  PROC DrawPart107()
    MoveL Offs(pOrigin,356.52,241.10,0.00),v60,z0,tPen\WObj:=wPaper;
    MoveL Offs(pOrigin,353.06,244.55,0.00),v40,z0,tPen\WObj:=wPaper;
    MoveL Offs(pOrigin,352.89,244.16,0.00),v40,z0,tPen\WObj:=wPaper;
    MoveL Offs(pOrigin,351.08,242.36,0.00),v40,z0,tPen\WObj:=wPaper;
    MoveL Offs(pOrigin,351.27,241.86,0.00),v40,z0,tPen\WObj:=wPaper;
    MoveL Offs(pOrigin,347.97,245.17,0.00),v40,z0,tPen\WObj:=wPaper;
    MoveL Offs(pOrigin,347.50,244.74,0.00),v40,z0,tPen\WObj:=wPaper;
    MoveL Offs(pOrigin,345.69,242.94,0.00),v40,z0,tPen\WObj:=wPaper;
    MoveL Offs(pOrigin,346.48,242.18,0.00),v40,z0,tPen\WObj:=wPaper;
    MoveL Offs(pOrigin,343.17,245.48,0.00),v40,z0,tPen\WObj:=wPaper;
    MoveL Offs(pOrigin,343.30,245.03,0.00),v40,z0,tPen\WObj:=wPaper;
    MoveL Offs(pOrigin,341.65,243.38,0.00),v40,z0,tPen\WObj:=wPaper;
    MoveL Offs(pOrigin,341.53,242.64,0.00),v40,z0,tPen\WObj:=wPaper;
    MoveL Offs(pOrigin,338.23,245.95,0.00),v40,z0,tPen\WObj:=wPaper;
    MoveL Offs(pOrigin,338.06,245.76,0.00),v40,z0,tPen\WObj:=wPaper;
    MoveL Offs(pOrigin,336.26,243.96,0.00),v40,z0,tPen\WObj:=wPaper;
    MoveL Offs(pOrigin,336.59,243.10,0.00),v40,z0,tPen\WObj:=wPaper;
    MoveL Offs(pOrigin,333.58,246.11,0.00),v40,z0,tPen\WObj:=wPaper;
    MoveL Offs(pOrigin,333.72,245.90,0.00),v40,z0,tPen\WObj:=wPaper;
    MoveL Offs(pOrigin,331.91,244.10,0.00),v40,z0,tPen\WObj:=wPaper;
    MoveL Offs(pOrigin,331.64,243.57,0.00),v40,z0,tPen\WObj:=wPaper;
    MoveL Offs(pOrigin,328.64,246.57,0.00),v40,z0,tPen\WObj:=wPaper;
    MoveL Offs(pOrigin,328.18,246.33,0.00),v40,z0,tPen\WObj:=wPaper;
    MoveL Offs(pOrigin,326.37,244.53,0.00),v40,fine,tPen\WObj:=wPaper;
    MoveL Offs(pOrigin,326.37,244.53,6.00),v60,z5,tPen\WObj:=wPaper;
    MoveL Offs(pOrigin,325.18,246.32,6.00),vTravel,z5,tPen\WObj:=wPaper;
    MoveL Offs(pOrigin,325.18,246.32,0.00),v60,z0,tPen\WObj:=wPaper;
    MoveL Offs(pOrigin,323.38,244.52,0.00),v40,z0,tPen\WObj:=wPaper;
    MoveL Offs(pOrigin,324.00,243.74,0.00),v40,z0,tPen\WObj:=wPaper;
    MoveL Offs(pOrigin,320.70,247.05,0.00),v40,z0,tPen\WObj:=wPaper;
    MoveL Offs(pOrigin,320.84,246.46,0.00),v40,z0,tPen\WObj:=wPaper;
    MoveL Offs(pOrigin,319.18,244.81,0.00),v40,z0,tPen\WObj:=wPaper;
    MoveL Offs(pOrigin,319.36,243.91,0.00),v40,z0,tPen\WObj:=wPaper;
    MoveL Offs(pOrigin,316.20,247.06,0.00),v40,z0,tPen\WObj:=wPaper;
    MoveL Offs(pOrigin,316.64,246.75,0.00),v40,z0,tPen\WObj:=wPaper;
    MoveL Offs(pOrigin,314.69,244.79,0.00),v40,z0,tPen\WObj:=wPaper;
    MoveL Offs(pOrigin,314.56,244.22,0.00),v40,z0,tPen\WObj:=wPaper;
    MoveL Offs(pOrigin,311.56,247.23,0.00),v40,z0,tPen\WObj:=wPaper;
    MoveL Offs(pOrigin,312.15,246.73,0.00),v40,z0,tPen\WObj:=wPaper;
    MoveL Offs(pOrigin,310.35,244.93,0.00),v40,z0,tPen\WObj:=wPaper;
    MoveL Offs(pOrigin,310.07,244.23,0.00),v40,z0,tPen\WObj:=wPaper;
    MoveL Offs(pOrigin,307.06,247.24,0.00),v40,z0,tPen\WObj:=wPaper;
    MoveL Offs(pOrigin,307.66,246.72,0.00),v40,z0,tPen\WObj:=wPaper;
    MoveL Offs(pOrigin,305.85,244.92,0.00),v40,z0,tPen\WObj:=wPaper;
    MoveL Offs(pOrigin,305.58,244.25,0.00),v40,z0,tPen\WObj:=wPaper;
    MoveL Offs(pOrigin,302.57,247.25,0.00),v40,z0,tPen\WObj:=wPaper;
    MoveL Offs(pOrigin,303.16,246.70,0.00),v40,z0,tPen\WObj:=wPaper;
    MoveL Offs(pOrigin,301.21,244.75,0.00),v40,z0,tPen\WObj:=wPaper;
    MoveL Offs(pOrigin,301.08,244.26,0.00),v40,z0,tPen\WObj:=wPaper;
    MoveL Offs(pOrigin,297.32,248.02,0.00),v40,z0,tPen\WObj:=wPaper;
    MoveL Offs(pOrigin,297.77,247.29,0.00),v40,z0,tPen\WObj:=wPaper;
    MoveL Offs(pOrigin,300.17,249.69,0.00),v40,z0,tPen\WObj:=wPaper;
    MoveL Offs(pOrigin,300.62,249.21,0.00),v40,z0,tPen\WObj:=wPaper;
    MoveL Offs(pOrigin,296.41,253.41,0.00),v40,z0,tPen\WObj:=wPaper;
    MoveL Offs(pOrigin,296.86,254.46,0.00),v40,z0,tPen\WObj:=wPaper;
    MoveL Offs(pOrigin,300.76,250.56,0.00),v40,z0,tPen\WObj:=wPaper;
    MoveL Offs(pOrigin,300.63,251.64,0.00),v40,z0,tPen\WObj:=wPaper;
    MoveL Offs(pOrigin,298.23,249.24,0.00),v40,fine,tPen\WObj:=wPaper;
    MoveL Offs(pOrigin,298.23,249.24,6.00),v60,z5,tPen\WObj:=wPaper;
    MoveL Offs(pOrigin,298.68,251.19,6.00),vTravel,z5,tPen\WObj:=wPaper;
    MoveL Offs(pOrigin,298.68,251.19,0.00),v60,z0,tPen\WObj:=wPaper;
    MoveL Offs(pOrigin,301.09,253.59,0.00),v40,z0,tPen\WObj:=wPaper;
    MoveL Offs(pOrigin,301.20,253.10,0.00),v40,z0,tPen\WObj:=wPaper;
    MoveL Offs(pOrigin,297.15,257.16,0.00),v40,z0,tPen\WObj:=wPaper;
    MoveL Offs(pOrigin,297.80,257.77,0.00),v40,z0,tPen\WObj:=wPaper;
    MoveL Offs(pOrigin,298.55,258.52,0.00),v40,z0,tPen\WObj:=wPaper;
    MoveL Offs(pOrigin,298.24,258.51,0.00),v40,z0,tPen\WObj:=wPaper;
    MoveL Offs(pOrigin,297.81,258.09,0.00),v40,z0,tPen\WObj:=wPaper;
    MoveL Offs(pOrigin,298.02,256.60,0.00),v40,fine,tPen\WObj:=wPaper;
    MoveL Offs(pOrigin,298.02,256.60,6.00),v60,z5,tPen\WObj:=wPaper;
    MoveL Offs(pOrigin,297.15,255.66,6.00),vTravel,z5,tPen\WObj:=wPaper;
    MoveL Offs(pOrigin,297.15,255.66,0.00),v60,z0,tPen\WObj:=wPaper;
    MoveL Offs(pOrigin,301.06,251.75,0.00),v40,fine,tPen\WObj:=wPaper;
    MoveL Offs(pOrigin,301.06,251.75,6.00),v60,z5,tPen\WObj:=wPaper;
    MoveL Offs(pOrigin,301.65,254.15,6.00),vTravel,z5,tPen\WObj:=wPaper;
    MoveL Offs(pOrigin,301.65,254.15,0.00),v60,z0,tPen\WObj:=wPaper;
    MoveL Offs(pOrigin,297.14,258.66,0.00),v40,fine,tPen\WObj:=wPaper;
    MoveL Offs(pOrigin,297.14,258.66,6.00),v60,z5,tPen\WObj:=wPaper;
    MoveL Offs(pOrigin,297.14,260.15,6.00),vTravel,z5,tPen\WObj:=wPaper;
    MoveL Offs(pOrigin,297.14,260.15,0.00),v60,z0,tPen\WObj:=wPaper;
    MoveL Offs(pOrigin,301.80,255.50,0.00),v40,z0,tPen\WObj:=wPaper;
    MoveL Offs(pOrigin,301.09,255.09,0.00),v40,z0,tPen\WObj:=wPaper;
    MoveL Offs(pOrigin,298.69,252.68,0.00),v40,fine,tPen\WObj:=wPaper;
    MoveL Offs(pOrigin,298.69,252.68,6.00),v60,z5,tPen\WObj:=wPaper;
    MoveL Offs(pOrigin,299.14,254.63,6.00),vTravel,z5,tPen\WObj:=wPaper;
    MoveL Offs(pOrigin,299.14,254.63,0.00),v60,z0,tPen\WObj:=wPaper;
    MoveL Offs(pOrigin,301.70,257.19,0.00),v40,z0,tPen\WObj:=wPaper;
    MoveL Offs(pOrigin,302.24,256.54,0.00),v40,z0,tPen\WObj:=wPaper;
    MoveL Offs(pOrigin,296.83,261.95,0.00),v40,fine,tPen\WObj:=wPaper;
    MoveL Offs(pOrigin,296.83,261.95,6.00),v60,z5,tPen\WObj:=wPaper;
    MoveL Offs(pOrigin,296.53,263.75,6.00),vTravel,z5,tPen\WObj:=wPaper;
    MoveL Offs(pOrigin,296.53,263.75,0.00),v60,z0,tPen\WObj:=wPaper;
    MoveL Offs(pOrigin,302.54,257.74,0.00),v40,fine,tPen\WObj:=wPaper;
    MoveL Offs(pOrigin,302.54,257.74,6.00),v60,z5,tPen\WObj:=wPaper;
    MoveL Offs(pOrigin,302.83,258.94,6.00),vTravel,z5,tPen\WObj:=wPaper;
    MoveL Offs(pOrigin,302.83,258.94,0.00),v60,z0,tPen\WObj:=wPaper;
    MoveL Offs(pOrigin,298.93,262.84,0.00),v40,fine,tPen\WObj:=wPaper;
    MoveL Offs(pOrigin,298.93,262.84,6.00),v60,z5,tPen\WObj:=wPaper;
    MoveL Offs(pOrigin,299.22,264.04,6.00),vTravel,z5,tPen\WObj:=wPaper;
    MoveL Offs(pOrigin,299.22,264.04,0.00),v60,z0,tPen\WObj:=wPaper;
    MoveL Offs(pOrigin,303.28,259.98,0.00),v40,z0,tPen\WObj:=wPaper;
    MoveL Offs(pOrigin,302.45,259.44,0.00),v40,z0,tPen\WObj:=wPaper;
    MoveL Offs(pOrigin,299.60,256.58,0.00),v40,fine,tPen\WObj:=wPaper;
    MoveL Offs(pOrigin,299.60,256.58,6.00),v60,z5,tPen\WObj:=wPaper;
    MoveL Offs(pOrigin,300.35,258.83,6.00),vTravel,z5,tPen\WObj:=wPaper;
    MoveL Offs(pOrigin,300.35,258.83,0.00),v60,z0,tPen\WObj:=wPaper;
    MoveL Offs(pOrigin,303.06,261.53,0.00),v40,z0,tPen\WObj:=wPaper;
    MoveL Offs(pOrigin,303.58,261.18,0.00),v40,z0,tPen\WObj:=wPaper;
    MoveL Offs(pOrigin,298.77,265.99,0.00),v40,fine,tPen\WObj:=wPaper;
    MoveL Offs(pOrigin,298.77,265.99,6.00),v60,z5,tPen\WObj:=wPaper;
    MoveL Offs(pOrigin,297.42,264.35,6.00),vTravel,z5,tPen\WObj:=wPaper;
    MoveL Offs(pOrigin,297.42,264.35,0.00),v60,z0,tPen\WObj:=wPaper;
    MoveL Offs(pOrigin,296.52,265.25,0.00),v40,fine,tPen\WObj:=wPaper;
    MoveL Offs(pOrigin,296.52,265.25,6.00),v60,z5,tPen\WObj:=wPaper;
    MoveL Offs(pOrigin,295.69,268.08,6.00),vTravel,z5,tPen\WObj:=wPaper;
    MoveL Offs(pOrigin,295.69,268.08,0.00),v60,z0,tPen\WObj:=wPaper;
    MoveL Offs(pOrigin,297.95,260.21,0.00),v40,z0,tPen\WObj:=wPaper;
    MoveL Offs(pOrigin,298.45,259.79,0.00),v40,fine,tPen\WObj:=wPaper;
    MoveL Offs(pOrigin,298.45,259.79,6.00),v60,z5,tPen\WObj:=wPaper;
    MoveL Offs(pOrigin,301.11,261.08,6.00),vTravel,z5,tPen\WObj:=wPaper;
  ENDPROC

  PROC DrawPart108()
    MoveL Offs(pOrigin,301.11,261.08,0.00),v60,z0,tPen\WObj:=wPaper;
    MoveL Offs(pOrigin,303.21,263.18,0.00),v40,z0,tPen\WObj:=wPaper;
    MoveL Offs(pOrigin,303.72,262.53,0.00),v40,z0,tPen\WObj:=wPaper;
    MoveL Offs(pOrigin,297.86,268.39,0.00),v40,fine,tPen\WObj:=wPaper;
    MoveL Offs(pOrigin,297.86,268.39,6.00),v60,z5,tPen\WObj:=wPaper;
    MoveL Offs(pOrigin,296.51,269.74,6.00),vTravel,z5,tPen\WObj:=wPaper;
    MoveL Offs(pOrigin,296.51,269.74,0.00),v60,z0,tPen\WObj:=wPaper;
    MoveL Offs(pOrigin,294.56,271.70,0.00),v40,z0,tPen\WObj:=wPaper;
    MoveL Offs(pOrigin,293.80,272.45,0.00),v40,z0,tPen\WObj:=wPaper;
    MoveL Offs(pOrigin,278.33,287.92,0.00),v40,fine,tPen\WObj:=wPaper;
    MoveL Offs(pOrigin,278.33,287.92,6.00),v60,z5,tPen\WObj:=wPaper;
    MoveL Offs(pOrigin,278.62,289.12,6.00),vTravel,z5,tPen\WObj:=wPaper;
    MoveL Offs(pOrigin,278.62,289.12,0.00),v60,z0,tPen\WObj:=wPaper;
    MoveL Offs(pOrigin,294.70,273.04,0.00),v40,fine,tPen\WObj:=wPaper;
    MoveL Offs(pOrigin,294.70,273.04,6.00),v60,z5,tPen\WObj:=wPaper;
    MoveL Offs(pOrigin,295.90,273.34,6.00),vTravel,z5,tPen\WObj:=wPaper;
    MoveL Offs(pOrigin,295.90,273.34,0.00),v60,z0,tPen\WObj:=wPaper;
    MoveL Offs(pOrigin,278.62,290.62,0.00),v40,z0,tPen\WObj:=wPaper;
    MoveL Offs(pOrigin,279.63,290.37,0.00),v40,z0,tPen\WObj:=wPaper;
    MoveL Offs(pOrigin,286.24,296.99,0.00),v40,z0,tPen\WObj:=wPaper;
    MoveL Offs(pOrigin,285.27,297.19,0.00),v40,z0,tPen\WObj:=wPaper;
    MoveL Offs(pOrigin,283.58,297.19,0.00),v40,z0,tPen\WObj:=wPaper;
    MoveL Offs(pOrigin,283.58,297.19,0.00),v40,z0,tPen\WObj:=wPaper;
    MoveL Offs(pOrigin,282.09,300.38,0.00),v40,z0,tPen\WObj:=wPaper;
    MoveL Offs(pOrigin,282.73,300.59,0.00),v40,z0,tPen\WObj:=wPaper;
    MoveL Offs(pOrigin,285.70,298.04,0.00),v40,z0,tPen\WObj:=wPaper;
    MoveL Offs(pOrigin,285.27,297.19,0.00),v40,z0,tPen\WObj:=wPaper;
    MoveL Offs(pOrigin,285.70,295.06,0.00),v40,z0,tPen\WObj:=wPaper;
    MoveL Offs(pOrigin,287.19,294.42,0.00),v40,z0,tPen\WObj:=wPaper;
    MoveL Offs(pOrigin,287.19,294.42,0.00),v40,z0,tPen\WObj:=wPaper;
    MoveL Offs(pOrigin,288.89,295.06,0.00),v40,z0,tPen\WObj:=wPaper;
    MoveL Offs(pOrigin,289.31,295.06,0.00),v40,z0,tPen\WObj:=wPaper;
    MoveL Offs(pOrigin,289.52,294.42,0.00),v40,z0,tPen\WObj:=wPaper;
    MoveL Offs(pOrigin,290.59,294.42,0.00),v40,fine,tPen\WObj:=wPaper;
    MoveL Offs(pOrigin,290.59,294.42,6.00),v60,z5,tPen\WObj:=wPaper;
    MoveL Offs(pOrigin,290.16,295.70,6.00),vTravel,z5,tPen\WObj:=wPaper;
    MoveL Offs(pOrigin,290.16,295.70,0.00),v60,z0,tPen\WObj:=wPaper;
    MoveL Offs(pOrigin,289.31,295.06,0.00),v40,fine,tPen\WObj:=wPaper;
    MoveL Offs(pOrigin,289.31,295.06,6.00),v60,z5,tPen\WObj:=wPaper;
    MoveL Offs(pOrigin,290.80,295.90,6.00),vTravel,z5,tPen\WObj:=wPaper;
    MoveL Offs(pOrigin,290.80,295.90,0.00),v60,z0,tPen\WObj:=wPaper;
    MoveL Offs(pOrigin,297.18,295.90,0.00),v40,z0,tPen\WObj:=wPaper;
    MoveL Offs(pOrigin,297.62,296.42,0.00),v40,z0,tPen\WObj:=wPaper;
    MoveL Offs(pOrigin,280.19,278.99,0.00),v40,z0,tPen\WObj:=wPaper;
    MoveL Offs(pOrigin,280.91,278.91,0.00),v40,z0,tPen\WObj:=wPaper;
    MoveL Offs(pOrigin,280.91,281.25,0.00),v40,z0,tPen\WObj:=wPaper;
    MoveL Offs(pOrigin,280.60,282.17,0.00),v40,z0,tPen\WObj:=wPaper;
    MoveL Offs(pOrigin,288.68,282.17,0.00),v40,fine,tPen\WObj:=wPaper;
    MoveL Offs(pOrigin,288.68,282.17,6.00),v60,z5,tPen\WObj:=wPaper;
    MoveL Offs(pOrigin,287.25,281.04,6.00),vTravel,z5,tPen\WObj:=wPaper;
    MoveL Offs(pOrigin,287.25,281.04,0.00),v60,z0,tPen\WObj:=wPaper;
    MoveL Offs(pOrigin,287.25,279.76,0.00),v40,z0,tPen\WObj:=wPaper;
    MoveL Offs(pOrigin,286.98,279.00,0.00),v40,z0,tPen\WObj:=wPaper;
    MoveL Offs(pOrigin,291.44,279.00,0.00),v40,fine,tPen\WObj:=wPaper;
    MoveL Offs(pOrigin,291.44,279.00,6.00),v60,z5,tPen\WObj:=wPaper;
    MoveL Offs(pOrigin,292.50,278.27,6.00),vTravel,z5,tPen\WObj:=wPaper;
    MoveL Offs(pOrigin,292.50,278.27,0.00),v60,z0,tPen\WObj:=wPaper;
    MoveL Offs(pOrigin,291.86,277.28,0.00),v40,z0,tPen\WObj:=wPaper;
    MoveL Offs(pOrigin,290.16,277.00,0.00),v40,z0,tPen\WObj:=wPaper;
    MoveL Offs(pOrigin,290.38,276.36,0.00),v40,z0,tPen\WObj:=wPaper;
    MoveL Offs(pOrigin,291.01,276.15,0.00),v40,z0,tPen\WObj:=wPaper;
    MoveL Offs(pOrigin,291.47,276.58,0.00),v40,z0,tPen\WObj:=wPaper;
    MoveL Offs(pOrigin,291.47,275.09,0.00),v40,z0,tPen\WObj:=wPaper;
    MoveL Offs(pOrigin,291.47,274.02,0.00),v40,z0,tPen\WObj:=wPaper;
    MoveL Offs(pOrigin,291.47,272.32,0.00),v40,z0,tPen\WObj:=wPaper;
    MoveL Offs(pOrigin,291.44,271.61,0.00),v40,z0,tPen\WObj:=wPaper;
    MoveL Offs(pOrigin,283.58,271.61,0.00),v40,z0,tPen\WObj:=wPaper;
    MoveL Offs(pOrigin,283.15,272.33,0.00),v40,z0,tPen\WObj:=wPaper;
    MoveL Offs(pOrigin,282.09,273.17,0.00),v40,z0,tPen\WObj:=wPaper;
    MoveL Offs(pOrigin,282.09,273.17,0.00),v40,z0,tPen\WObj:=wPaper;
    MoveL Offs(pOrigin,280.39,273.17,0.00),v40,z0,tPen\WObj:=wPaper;
    MoveL Offs(pOrigin,279.75,272.75,0.00),v40,z0,tPen\WObj:=wPaper;
    MoveL Offs(pOrigin,280.17,273.00,0.00),v40,z0,tPen\WObj:=wPaper;
    MoveL Offs(pOrigin,275.82,268.64,0.00),v40,z0,tPen\WObj:=wPaper;
    MoveL Offs(pOrigin,275.24,268.61,0.00),v40,z0,tPen\WObj:=wPaper;
    MoveL Offs(pOrigin,277.49,266.36,0.00),v40,fine,tPen\WObj:=wPaper;
    MoveL Offs(pOrigin,277.49,266.36,6.00),v60,z5,tPen\WObj:=wPaper;
    MoveL Offs(pOrigin,277.64,267.70,6.00),vTravel,z5,tPen\WObj:=wPaper;
    MoveL Offs(pOrigin,277.64,267.70,0.00),v60,z0,tPen\WObj:=wPaper;
    MoveL Offs(pOrigin,274.79,270.56,0.00),v40,z0,tPen\WObj:=wPaper;
    MoveL Offs(pOrigin,275.50,271.48,0.00),v40,z0,tPen\WObj:=wPaper;
    MoveL Offs(pOrigin,274.86,271.90,0.00),v40,z0,tPen\WObj:=wPaper;
    MoveL Offs(pOrigin,274.44,273.39,0.00),v40,z0,tPen\WObj:=wPaper;
    MoveL Offs(pOrigin,274.44,273.39,0.00),v40,z0,tPen\WObj:=wPaper;
    MoveL Offs(pOrigin,272.10,274.45,0.00),v40,z0,tPen\WObj:=wPaper;
    MoveL Offs(pOrigin,270.40,274.66,0.00),v40,z0,tPen\WObj:=wPaper;
    MoveL Offs(pOrigin,269.76,274.38,0.00),v40,z0,tPen\WObj:=wPaper;
    MoveL Offs(pOrigin,268.49,274.45,0.00),v40,z0,tPen\WObj:=wPaper;
    MoveL Offs(pOrigin,268.49,274.45,0.00),v40,z0,tPen\WObj:=wPaper;
    MoveL Offs(pOrigin,267.64,275.44,0.00),v40,z0,tPen\WObj:=wPaper;
    MoveL Offs(pOrigin,264.45,276.36,0.00),v40,z0,tPen\WObj:=wPaper;
    MoveL Offs(pOrigin,264.45,276.36,0.00),v40,z0,tPen\WObj:=wPaper;
    MoveL Offs(pOrigin,264.02,277.00,0.00),v40,z0,tPen\WObj:=wPaper;
    MoveL Offs(pOrigin,263.39,277.00,0.00),v40,z0,tPen\WObj:=wPaper;
    MoveL Offs(pOrigin,263.17,276.36,0.00),v40,z0,tPen\WObj:=wPaper;
    MoveL Offs(pOrigin,263.17,276.36,0.00),v40,z0,tPen\WObj:=wPaper;
    MoveL Offs(pOrigin,264.45,276.15,0.00),v40,z0,tPen\WObj:=wPaper;
    MoveL Offs(pOrigin,264.45,276.36,0.00),v40,z0,tPen\WObj:=wPaper;
    MoveL Offs(pOrigin,264.15,276.40,0.00),v40,z0,tPen\WObj:=wPaper;
    MoveL Offs(pOrigin,259.50,271.74,0.00),v40,fine,tPen\WObj:=wPaper;
    MoveL Offs(pOrigin,259.50,271.74,6.00),v60,z5,tPen\WObj:=wPaper;
    MoveL Offs(pOrigin,260.41,272.66,6.00),vTravel,z5,tPen\WObj:=wPaper;
    MoveL Offs(pOrigin,260.41,272.66,0.00),v60,z0,tPen\WObj:=wPaper;
    MoveL Offs(pOrigin,256.38,272.66,0.00),v40,z0,tPen\WObj:=wPaper;
    MoveL Offs(pOrigin,256.38,271.61,0.00),v40,z0,tPen\WObj:=wPaper;
    MoveL Offs(pOrigin,253.19,271.61,0.00),v40,z0,tPen\WObj:=wPaper;
    MoveL Offs(pOrigin,253.40,272.66,0.00),v40,z0,tPen\WObj:=wPaper;
    MoveL Offs(pOrigin,249.36,272.66,0.00),v40,z0,tPen\WObj:=wPaper;
    MoveL Offs(pOrigin,249.15,272.75,0.00),v40,z0,tPen\WObj:=wPaper;
    MoveL Offs(pOrigin,249.79,272.18,0.00),v40,z0,tPen\WObj:=wPaper;
    MoveL Offs(pOrigin,250.43,272.11,0.00),v40,z0,tPen\WObj:=wPaper;
    MoveL Offs(pOrigin,259.35,274.24,0.00),v40,z0,tPen\WObj:=wPaper;
    MoveL Offs(pOrigin,262.33,274.66,0.00),v40,z0,tPen\WObj:=wPaper;
    MoveL Offs(pOrigin,265.73,274.45,0.00),v40,z0,tPen\WObj:=wPaper;
    MoveL Offs(pOrigin,265.73,274.45,0.00),v40,z0,tPen\WObj:=wPaper;
    MoveL Offs(pOrigin,266.58,274.66,0.00),v40,z0,tPen\WObj:=wPaper;
    MoveL Offs(pOrigin,266.79,275.51,0.00),v40,z0,tPen\WObj:=wPaper;
    MoveL Offs(pOrigin,266.40,275.65,0.00),v40,z0,tPen\WObj:=wPaper;
    MoveL Offs(pOrigin,263.39,272.65,0.00),v40,z0,tPen\WObj:=wPaper;
    MoveL Offs(pOrigin,263.10,271.79,0.00),v40,z0,tPen\WObj:=wPaper;
  ENDPROC

  PROC DrawPart109()
    MoveL Offs(pOrigin,258.89,276.00,0.00),v40,z0,tPen\WObj:=wPaper;
    MoveL Offs(pOrigin,259.21,275.93,0.00),v40,z0,tPen\WObj:=wPaper;
    MoveL Offs(pOrigin,252.60,269.32,0.00),v40,z0,tPen\WObj:=wPaper;
    MoveL Offs(pOrigin,252.12,268.29,0.00),v40,z0,tPen\WObj:=wPaper;
    MoveL Offs(pOrigin,252.55,268.71,0.00),v40,z0,tPen\WObj:=wPaper;
    MoveL Offs(pOrigin,252.12,268.29,0.00),v40,z0,tPen\WObj:=wPaper;
    MoveL Offs(pOrigin,251.42,268.53,0.00),v40,z0,tPen\WObj:=wPaper;
    MoveL Offs(pOrigin,256.83,263.12,0.00),v40,fine,tPen\WObj:=wPaper;
    MoveL Offs(pOrigin,256.83,263.12,6.00),v60,z5,tPen\WObj:=wPaper;
    MoveL Offs(pOrigin,258.33,263.12,6.00),vTravel,z5,tPen\WObj:=wPaper;
    MoveL Offs(pOrigin,258.33,263.12,0.00),v60,z0,tPen\WObj:=wPaper;
    MoveL Offs(pOrigin,247.06,274.39,0.00),v40,z0,tPen\WObj:=wPaper;
    MoveL Offs(pOrigin,246.31,273.64,0.00),v40,z0,tPen\WObj:=wPaper;
    MoveL Offs(pOrigin,250.22,269.73,0.00),v40,z0,tPen\WObj:=wPaper;
    MoveL Offs(pOrigin,249.17,269.29,0.00),v40,z0,tPen\WObj:=wPaper;
    MoveL Offs(pOrigin,245.87,272.59,0.00),v40,z0,tPen\WObj:=wPaper;
    MoveL Offs(pOrigin,246.81,272.96,0.00),v40,z0,tPen\WObj:=wPaper;
    MoveL Offs(pOrigin,247.24,273.60,0.00),v40,z0,tPen\WObj:=wPaper;
    MoveL Offs(pOrigin,248.73,274.24,0.00),v40,z0,tPen\WObj:=wPaper;
    MoveL Offs(pOrigin,249.15,274.24,0.00),v40,z0,tPen\WObj:=wPaper;
    MoveL Offs(pOrigin,250.21,275.09,0.00),v40,z0,tPen\WObj:=wPaper;
    MoveL Offs(pOrigin,250.85,275.09,0.00),v40,z0,tPen\WObj:=wPaper;
    MoveL Offs(pOrigin,251.06,274.45,0.00),v40,z0,tPen\WObj:=wPaper;
    MoveL Offs(pOrigin,251.06,274.45,0.00),v40,z0,tPen\WObj:=wPaper;
    MoveL Offs(pOrigin,250.21,273.81,0.00),v40,z0,tPen\WObj:=wPaper;
    MoveL Offs(pOrigin,249.15,273.60,0.00),v40,z0,tPen\WObj:=wPaper;
    MoveL Offs(pOrigin,249.15,272.75,0.00),v40,z0,tPen\WObj:=wPaper;
    MoveL Offs(pOrigin,248.73,272.11,0.00),v40,z0,tPen\WObj:=wPaper;
    MoveL Offs(pOrigin,248.94,271.05,0.00),v40,z0,tPen\WObj:=wPaper;
    MoveL Offs(pOrigin,250.64,270.62,0.00),v40,z0,tPen\WObj:=wPaper;
    MoveL Offs(pOrigin,251.27,270.84,0.00),v40,z0,tPen\WObj:=wPaper;
    MoveL Offs(pOrigin,251.27,270.84,0.00),v40,z0,tPen\WObj:=wPaper;
    MoveL Offs(pOrigin,251.91,271.62,0.00),v40,z0,tPen\WObj:=wPaper;
    MoveL Offs(pOrigin,254.25,272.33,0.00),v40,z0,tPen\WObj:=wPaper;
    MoveL Offs(pOrigin,262.33,273.81,0.00),v40,z0,tPen\WObj:=wPaper;
    MoveL Offs(pOrigin,265.09,273.81,0.00),v40,z0,tPen\WObj:=wPaper;
    MoveL Offs(pOrigin,265.73,274.45,0.00),v40,z0,tPen\WObj:=wPaper;
    MoveL Offs(pOrigin,265.09,274.78,0.00),v40,z0,tPen\WObj:=wPaper;
    MoveL Offs(pOrigin,255.74,274.78,0.00),v40,z0,tPen\WObj:=wPaper;
    MoveL Offs(pOrigin,255.76,275.47,0.00),v40,z0,tPen\WObj:=wPaper;
    MoveL Offs(pOrigin,250.95,270.66,0.00),v40,z0,tPen\WObj:=wPaper;
    MoveL Offs(pOrigin,251.27,270.84,0.00),v40,z0,tPen\WObj:=wPaper;
    MoveL Offs(pOrigin,254.04,270.62,0.00),v40,z0,tPen\WObj:=wPaper;
    MoveL Offs(pOrigin,254.04,270.20,0.00),v40,z0,tPen\WObj:=wPaper;
    MoveL Offs(pOrigin,250.78,267.01,0.00),v40,z0,tPen\WObj:=wPaper;
    MoveL Offs(pOrigin,250.43,266.16,0.00),v40,z0,tPen\WObj:=wPaper;
    MoveL Offs(pOrigin,250.64,265.74,0.00),v40,z0,tPen\WObj:=wPaper;
    MoveL Offs(pOrigin,250.64,265.74,0.00),v40,z0,tPen\WObj:=wPaper;
    MoveL Offs(pOrigin,251.91,266.02,0.00),v40,z0,tPen\WObj:=wPaper;
    MoveL Offs(pOrigin,252.55,267.44,0.00),v40,z0,tPen\WObj:=wPaper;
    MoveL Offs(pOrigin,253.19,267.93,0.00),v40,z0,tPen\WObj:=wPaper;
    MoveL Offs(pOrigin,254.25,268.08,0.00),v40,z0,tPen\WObj:=wPaper;
    MoveL Offs(pOrigin,254.04,267.65,0.00),v40,z0,tPen\WObj:=wPaper;
    MoveL Offs(pOrigin,254.25,268.08,0.00),v40,z0,tPen\WObj:=wPaper;
    MoveL Offs(pOrigin,254.04,267.65,0.00),v40,fine,tPen\WObj:=wPaper;
    MoveL Offs(pOrigin,254.04,267.65,6.00),v60,z5,tPen\WObj:=wPaper;
    MoveL Offs(pOrigin,253.82,269.56,6.00),vTravel,z5,tPen\WObj:=wPaper;
    MoveL Offs(pOrigin,253.82,269.56,0.00),v60,z0,tPen\WObj:=wPaper;
    MoveL Offs(pOrigin,254.46,268.29,0.00),v40,z0,tPen\WObj:=wPaper;
    MoveL Offs(pOrigin,253.82,266.80,0.00),v40,z0,tPen\WObj:=wPaper;
    MoveL Offs(pOrigin,253.19,266.23,0.00),v40,z0,tPen\WObj:=wPaper;
    MoveL Offs(pOrigin,252.12,265.95,0.00),v40,z0,tPen\WObj:=wPaper;
    MoveL Offs(pOrigin,252.12,265.27,0.00),v40,z0,tPen\WObj:=wPaper;
    MoveL Offs(pOrigin,253.82,265.27,0.00),v40,z0,tPen\WObj:=wPaper;
    MoveL Offs(pOrigin,254.46,265.74,0.00),v40,z0,tPen\WObj:=wPaper;
    MoveL Offs(pOrigin,254.89,266.16,0.00),v40,z0,tPen\WObj:=wPaper;
    MoveL Offs(pOrigin,254.46,265.74,0.00),v40,z0,tPen\WObj:=wPaper;
    MoveL Offs(pOrigin,254.83,265.58,0.00),v40,z0,tPen\WObj:=wPaper;
    MoveL Offs(pOrigin,253.18,263.93,0.00),v40,z0,tPen\WObj:=wPaper;
    MoveL Offs(pOrigin,252.34,264.25,0.00),v40,z0,tPen\WObj:=wPaper;
    MoveL Offs(pOrigin,251.91,263.68,0.00),v40,z0,tPen\WObj:=wPaper;
    MoveL Offs(pOrigin,250.64,263.68,0.00),v40,z0,tPen\WObj:=wPaper;
    MoveL Offs(pOrigin,250.43,264.25,0.00),v40,z0,tPen\WObj:=wPaper;
    MoveL Offs(pOrigin,250.64,265.74,0.00),v40,z0,tPen\WObj:=wPaper;
    MoveL Offs(pOrigin,250.43,265.74,0.00),v40,z0,tPen\WObj:=wPaper;
    MoveL Offs(pOrigin,249.79,265.10,0.00),v40,z0,tPen\WObj:=wPaper;
    MoveL Offs(pOrigin,249.15,264.89,0.00),v40,z0,tPen\WObj:=wPaper;
    MoveL Offs(pOrigin,250.21,265.74,0.00),v40,z0,tPen\WObj:=wPaper;
    MoveL Offs(pOrigin,250.21,265.74,0.00),v40,z0,tPen\WObj:=wPaper;
    MoveL Offs(pOrigin,249.15,266.66,0.00),v40,z0,tPen\WObj:=wPaper;
    MoveL Offs(pOrigin,248.58,266.73,0.00),v40,z0,tPen\WObj:=wPaper;
    MoveL Offs(pOrigin,248.30,265.52,0.00),v40,z0,tPen\WObj:=wPaper;
    MoveL Offs(pOrigin,249.15,264.89,0.00),v40,z0,tPen\WObj:=wPaper;
    MoveL Offs(pOrigin,249.15,264.89,0.00),v40,z0,tPen\WObj:=wPaper;
    MoveL Offs(pOrigin,247.88,262.76,0.00),v40,z0,tPen\WObj:=wPaper;
    MoveL Offs(pOrigin,248.73,261.06,0.00),v40,z0,tPen\WObj:=wPaper;
    MoveL Offs(pOrigin,250.00,259.79,0.00),v40,z0,tPen\WObj:=wPaper;
    MoveL Offs(pOrigin,250.00,258.73,0.00),v40,z0,tPen\WObj:=wPaper;
    MoveL Offs(pOrigin,249.15,257.88,0.00),v40,z0,tPen\WObj:=wPaper;
    MoveL Offs(pOrigin,249.15,258.30,0.00),v40,z0,tPen\WObj:=wPaper;
    MoveL Offs(pOrigin,248.30,259.79,0.00),v40,z0,tPen\WObj:=wPaper;
    MoveL Offs(pOrigin,248.51,261.06,0.00),v40,fine,tPen\WObj:=wPaper;
    MoveL Offs(pOrigin,248.51,261.06,6.00),v60,z5,tPen\WObj:=wPaper;
    MoveL Offs(pOrigin,249.58,261.82,6.00),vTravel,z5,tPen\WObj:=wPaper;
    MoveL Offs(pOrigin,249.58,261.82,0.00),v60,z0,tPen\WObj:=wPaper;
    MoveL Offs(pOrigin,246.87,259.12,0.00),v40,z0,tPen\WObj:=wPaper;
    MoveL Offs(pOrigin,246.06,258.96,0.00),v40,z0,tPen\WObj:=wPaper;
    MoveL Offs(pOrigin,250.87,254.15,0.00),v40,fine,tPen\WObj:=wPaper;
    MoveL Offs(pOrigin,250.87,254.15,6.00),v60,z5,tPen\WObj:=wPaper;
    MoveL Offs(pOrigin,253.42,253.10,6.00),vTravel,z5,tPen\WObj:=wPaper;
    MoveL Offs(pOrigin,253.42,253.10,0.00),v60,z0,tPen\WObj:=wPaper;
    MoveL Offs(pOrigin,245.00,261.51,0.00),v40,z0,tPen\WObj:=wPaper;
    MoveL Offs(pOrigin,245.39,262.11,0.00),v40,z0,tPen\WObj:=wPaper;
    MoveL Offs(pOrigin,250.65,267.37,0.00),v40,z0,tPen\WObj:=wPaper;
    MoveL Offs(pOrigin,250.68,267.79,0.00),v40,z0,tPen\WObj:=wPaper;
    MoveL Offs(pOrigin,257.74,260.72,0.00),v40,fine,tPen\WObj:=wPaper;
    MoveL Offs(pOrigin,257.74,260.72,6.00),v60,z5,tPen\WObj:=wPaper;
    MoveL Offs(pOrigin,259.09,259.37,6.00),vTravel,z5,tPen\WObj:=wPaper;
    MoveL Offs(pOrigin,259.09,259.37,0.00),v60,z0,tPen\WObj:=wPaper;
    MoveL Offs(pOrigin,259.99,258.47,0.00),v40,z0,tPen\WObj:=wPaper;
    MoveL Offs(pOrigin,258.95,258.02,0.00),v40,z0,tPen\WObj:=wPaper;
    MoveL Offs(pOrigin,249.63,267.34,0.00),v40,fine,tPen\WObj:=wPaper;
    MoveL Offs(pOrigin,249.63,267.34,6.00),v60,z5,tPen\WObj:=wPaper;
    MoveL Offs(pOrigin,248.43,267.04,6.00),vTravel,z5,tPen\WObj:=wPaper;
    MoveL Offs(pOrigin,248.43,267.04,0.00),v60,z0,tPen\WObj:=wPaper;
    MoveL Offs(pOrigin,257.30,258.18,0.00),v40,fine,tPen\WObj:=wPaper;
    MoveL Offs(pOrigin,257.30,258.18,6.00),v60,z5,tPen\WObj:=wPaper;
    MoveL Offs(pOrigin,255.20,258.78,6.00),vTravel,z5,tPen\WObj:=wPaper;
    MoveL Offs(pOrigin,255.20,258.78,0.00),v60,z0,tPen\WObj:=wPaper;
    MoveL Offs(pOrigin,243.33,270.65,0.00),v40,fine,tPen\WObj:=wPaper;
  ENDPROC

  PROC DrawPart110()
    MoveL Offs(pOrigin,243.33,270.65,6.00),v60,z5,tPen\WObj:=wPaper;
    MoveL Offs(pOrigin,243.63,268.86,6.00),vTravel,z5,tPen\WObj:=wPaper;
    MoveL Offs(pOrigin,243.63,268.86,0.00),v60,z0,tPen\WObj:=wPaper;
    MoveL Offs(pOrigin,252.65,259.84,0.00),v40,fine,tPen\WObj:=wPaper;
    MoveL Offs(pOrigin,252.65,259.84,6.00),v60,z5,tPen\WObj:=wPaper;
    MoveL Offs(pOrigin,252.12,261.70,6.00),vTravel,z5,tPen\WObj:=wPaper;
    MoveL Offs(pOrigin,252.12,261.70,0.00),v60,z0,tPen\WObj:=wPaper;
    MoveL Offs(pOrigin,252.34,261.20,0.00),v40,z0,tPen\WObj:=wPaper;
    MoveL Offs(pOrigin,254.68,259.93,0.00),v40,z0,tPen\WObj:=wPaper;
    MoveL Offs(pOrigin,259.35,258.51,0.00),v40,z0,tPen\WObj:=wPaper;
    MoveL Offs(pOrigin,262.54,258.51,0.00),v40,fine,tPen\WObj:=wPaper;
    MoveL Offs(pOrigin,262.54,258.51,6.00),v60,z5,tPen\WObj:=wPaper;
    MoveL Offs(pOrigin,261.26,260.85,6.00),vTravel,z5,tPen\WObj:=wPaper;
    MoveL Offs(pOrigin,261.26,260.85,0.00),v60,z0,tPen\WObj:=wPaper;
    MoveL Offs(pOrigin,256.16,261.49,0.00),v40,z0,tPen\WObj:=wPaper;
    MoveL Offs(pOrigin,252.98,262.55,0.00),v40,z0,tPen\WObj:=wPaper;
    MoveL Offs(pOrigin,252.41,262.48,0.00),v40,z0,tPen\WObj:=wPaper;
    MoveL Offs(pOrigin,251.91,261.77,0.00),v40,z0,tPen\WObj:=wPaper;
    MoveL Offs(pOrigin,250.85,261.91,0.00),v40,fine,tPen\WObj:=wPaper;
    MoveL Offs(pOrigin,250.85,261.91,6.00),v60,z5,tPen\WObj:=wPaper;
    MoveL Offs(pOrigin,250.55,260.45,6.00),vTravel,z5,tPen\WObj:=wPaper;
    MoveL Offs(pOrigin,250.55,260.45,0.00),v60,z0,tPen\WObj:=wPaper;
    MoveL Offs(pOrigin,242.28,268.71,0.00),v40,z0,tPen\WObj:=wPaper;
    MoveL Offs(pOrigin,242.26,267.94,0.00),v40,z0,tPen\WObj:=wPaper;
    MoveL Offs(pOrigin,240.30,265.99,0.00),v40,z0,tPen\WObj:=wPaper;
    MoveL Offs(pOrigin,240.05,264.97,0.00),v40,z0,tPen\WObj:=wPaper;
    MoveL Offs(pOrigin,233.59,271.43,0.00),v40,z0,tPen\WObj:=wPaper;
    MoveL Offs(pOrigin,233.21,271.48,0.00),v40,z0,tPen\WObj:=wPaper;
    MoveL Offs(pOrigin,231.94,271.90,0.00),v40,z0,tPen\WObj:=wPaper;
    MoveL Offs(pOrigin,231.30,271.26,0.00),v40,z0,tPen\WObj:=wPaper;
    MoveL Offs(pOrigin,232.08,271.20,0.00),v40,z0,tPen\WObj:=wPaper;
    MoveL Offs(pOrigin,222.77,261.89,0.00),v40,z0,tPen\WObj:=wPaper;
    MoveL Offs(pOrigin,223.22,262.10,0.00),v40,z0,tPen\WObj:=wPaper;
    MoveL Offs(pOrigin,228.96,262.10,0.00),v40,z0,tPen\WObj:=wPaper;
    MoveL Offs(pOrigin,228.96,261.91,0.00),v40,z0,tPen\WObj:=wPaper;
    MoveL Offs(pOrigin,227.90,262.12,0.00),v40,z0,tPen\WObj:=wPaper;
    MoveL Offs(pOrigin,228.11,261.91,0.00),v40,z0,tPen\WObj:=wPaper;
    MoveL Offs(pOrigin,228.11,264.46,0.00),v40,z0,tPen\WObj:=wPaper;
    MoveL Offs(pOrigin,228.32,265.10,0.00),v40,z0,tPen\WObj:=wPaper;
    MoveL Offs(pOrigin,226.84,265.10,0.00),v40,z0,tPen\WObj:=wPaper;
    MoveL Offs(pOrigin,226.41,265.74,0.00),v40,z0,tPen\WObj:=wPaper;
    MoveL Offs(pOrigin,225.99,265.27,0.00),v40,z0,tPen\WObj:=wPaper;
    MoveL Offs(pOrigin,232.36,265.27,0.00),v40,z0,tPen\WObj:=wPaper;
    MoveL Offs(pOrigin,232.81,265.96,0.00),v40,z0,tPen\WObj:=wPaper;
    MoveL Offs(pOrigin,226.80,259.95,0.00),v40,z0,tPen\WObj:=wPaper;
    MoveL Offs(pOrigin,226.44,259.17,0.00),v40,z0,tPen\WObj:=wPaper;
    MoveL Offs(pOrigin,215.47,270.14,0.00),v40,z0,tPen\WObj:=wPaper;
    MoveL Offs(pOrigin,216.05,270.11,0.00),v40,z0,tPen\WObj:=wPaper;
    MoveL Offs(pOrigin,213.50,267.55,0.00),v40,z0,tPen\WObj:=wPaper;
    MoveL Offs(pOrigin,213.88,267.86,0.00),v40,z0,tPen\WObj:=wPaper;
    MoveL Offs(pOrigin,214.30,268.57,0.00),v40,z0,tPen\WObj:=wPaper;
    MoveL Offs(pOrigin,217.06,270.41,0.00),v40,z0,tPen\WObj:=wPaper;
    MoveL Offs(pOrigin,216.36,270.74,0.00),v40,z0,tPen\WObj:=wPaper;
    MoveL Offs(pOrigin,227.63,259.47,0.00),v40,fine,tPen\WObj:=wPaper;
    MoveL Offs(pOrigin,227.63,259.47,6.00),v60,z5,tPen\WObj:=wPaper;
    MoveL Offs(pOrigin,226.41,259.15,6.00),vTravel,z5,tPen\WObj:=wPaper;
    MoveL Offs(pOrigin,226.41,259.15,0.00),v60,z0,tPen\WObj:=wPaper;
    MoveL Offs(pOrigin,223.65,258.94,0.00),v40,z0,tPen\WObj:=wPaper;
    MoveL Offs(pOrigin,223.23,259.15,0.00),v40,z0,tPen\WObj:=wPaper;
    MoveL Offs(pOrigin,222.87,260.00,0.00),v40,z0,tPen\WObj:=wPaper;
    MoveL Offs(pOrigin,224.07,260.85,0.00),v40,z0,tPen\WObj:=wPaper;
    MoveL Offs(pOrigin,224.07,260.85,0.00),v40,z0,tPen\WObj:=wPaper;
    MoveL Offs(pOrigin,225.99,260.64,0.00),v40,z0,tPen\WObj:=wPaper;
    MoveL Offs(pOrigin,226.20,261.06,0.00),v40,z0,tPen\WObj:=wPaper;
    MoveL Offs(pOrigin,226.20,261.06,0.00),v40,z0,tPen\WObj:=wPaper;
    MoveL Offs(pOrigin,227.05,261.27,0.00),v40,z0,tPen\WObj:=wPaper;
    MoveL Offs(pOrigin,227.69,262.12,0.00),v40,z0,tPen\WObj:=wPaper;
    MoveL Offs(pOrigin,227.69,263.40,0.00),v40,fine,tPen\WObj:=wPaper;
    MoveL Offs(pOrigin,227.69,263.40,6.00),v60,z5,tPen\WObj:=wPaper;
    MoveL Offs(pOrigin,227.05,264.46,6.00),vTravel,z5,tPen\WObj:=wPaper;
    MoveL Offs(pOrigin,227.05,264.46,0.00),v60,z0,tPen\WObj:=wPaper;
    MoveL Offs(pOrigin,227.05,261.49,0.00),v40,z0,tPen\WObj:=wPaper;
    MoveL Offs(pOrigin,227.05,261.06,0.00),v40,z0,tPen\WObj:=wPaper;
    MoveL Offs(pOrigin,227.48,260.64,0.00),v40,z0,tPen\WObj:=wPaper;
    MoveL Offs(pOrigin,228.32,260.64,0.00),v40,z0,tPen\WObj:=wPaper;
    MoveL Offs(pOrigin,228.96,261.27,0.00),v40,z0,tPen\WObj:=wPaper;
    MoveL Offs(pOrigin,228.96,261.91,0.00),v40,z0,tPen\WObj:=wPaper;
    MoveL Offs(pOrigin,229.60,263.61,0.00),v40,z0,tPen\WObj:=wPaper;
    MoveL Offs(pOrigin,230.88,263.26,0.00),v40,z0,tPen\WObj:=wPaper;
    MoveL Offs(pOrigin,231.51,262.34,0.00),v40,z0,tPen\WObj:=wPaper;
    MoveL Offs(pOrigin,231.51,262.34,0.00),v40,z0,tPen\WObj:=wPaper;
    MoveL Offs(pOrigin,233.21,262.12,0.00),v40,z0,tPen\WObj:=wPaper;
    MoveL Offs(pOrigin,233.21,262.12,0.00),v40,z0,tPen\WObj:=wPaper;
    MoveL Offs(pOrigin,233.64,262.98,0.00),v40,z0,tPen\WObj:=wPaper;
    MoveL Offs(pOrigin,234.06,263.16,0.00),v40,z0,tPen\WObj:=wPaper;
    MoveL Offs(pOrigin,231.30,263.16,0.00),v40,z0,tPen\WObj:=wPaper;
    MoveL Offs(pOrigin,231.51,262.34,0.00),v40,z0,tPen\WObj:=wPaper;
    MoveL Offs(pOrigin,230.88,261.63,0.00),v40,z0,tPen\WObj:=wPaper;
    MoveL Offs(pOrigin,229.60,261.27,0.00),v40,z0,tPen\WObj:=wPaper;
    MoveL Offs(pOrigin,229.03,261.49,0.00),v40,z0,tPen\WObj:=wPaper;
    MoveL Offs(pOrigin,228.96,261.91,0.00),v40,z0,tPen\WObj:=wPaper;
    MoveL Offs(pOrigin,228.32,261.05,0.00),v40,z0,tPen\WObj:=wPaper;
    MoveL Offs(pOrigin,224.08,261.05,0.00),v40,z0,tPen\WObj:=wPaper;
    MoveL Offs(pOrigin,224.07,260.85,0.00),v40,z0,tPen\WObj:=wPaper;
    MoveL Offs(pOrigin,224.29,261.49,0.00),v40,z0,tPen\WObj:=wPaper;
    MoveL Offs(pOrigin,224.71,261.70,0.00),v40,z0,tPen\WObj:=wPaper;
    MoveL Offs(pOrigin,225.56,261.63,0.00),v40,z0,tPen\WObj:=wPaper;
    MoveL Offs(pOrigin,226.20,261.06,0.00),v40,z0,tPen\WObj:=wPaper;
    MoveL Offs(pOrigin,226.00,261.27,0.00),v40,z0,tPen\WObj:=wPaper;
    MoveL Offs(pOrigin,226.00,264.46,0.00),v40,z0,tPen\WObj:=wPaper;
    MoveL Offs(pOrigin,224.94,264.04,0.00),v40,z0,tPen\WObj:=wPaper;
    MoveL Offs(pOrigin,224.94,261.27,0.00),v40,z0,tPen\WObj:=wPaper;
    MoveL Offs(pOrigin,224.07,261.49,0.00),v40,z0,tPen\WObj:=wPaper;
    MoveL Offs(pOrigin,223.08,262.20,0.00),v40,z0,tPen\WObj:=wPaper;
    MoveL Offs(pOrigin,222.80,262.83,0.00),v40,z0,tPen\WObj:=wPaper;
    MoveL Offs(pOrigin,221.10,261.91,0.00),v40,z0,tPen\WObj:=wPaper;
    MoveL Offs(pOrigin,220.89,261.49,0.00),v40,z0,tPen\WObj:=wPaper;
    MoveL Offs(pOrigin,221.10,260.71,0.00),v40,z0,tPen\WObj:=wPaper;
    MoveL Offs(pOrigin,223.01,260.42,0.00),v40,z0,tPen\WObj:=wPaper;
    MoveL Offs(pOrigin,223.21,260.84,0.00),v40,z0,tPen\WObj:=wPaper;
    MoveL Offs(pOrigin,232.83,270.46,0.00),v40,z0,tPen\WObj:=wPaper;
    MoveL Offs(pOrigin,233.58,269.71,0.00),v40,z0,tPen\WObj:=wPaper;
    MoveL Offs(pOrigin,223.81,259.94,0.00),v40,z0,tPen\WObj:=wPaper;
    MoveL Offs(pOrigin,223.59,259.03,0.00),v40,z0,tPen\WObj:=wPaper;
    MoveL Offs(pOrigin,218.63,263.99,0.00),v40,z0,tPen\WObj:=wPaper;
    MoveL Offs(pOrigin,217.73,263.39,0.00),v40,z0,tPen\WObj:=wPaper;
    MoveL Offs(pOrigin,221.94,259.19,0.00),v40,z0,tPen\WObj:=wPaper;
    MoveL Offs(pOrigin,222.80,259.36,0.00),v40,z0,tPen\WObj:=wPaper;
    MoveL Offs(pOrigin,220.68,259.79,0.00),v40,z0,tPen\WObj:=wPaper;
    MoveL Offs(pOrigin,220.44,259.19,0.00),v40,z0,tPen\WObj:=wPaper;
  ENDPROC

  PROC DrawPart111()
    MoveL Offs(pOrigin,216.99,262.65,0.00),v40,z0,tPen\WObj:=wPaper;
    MoveL Offs(pOrigin,216.24,261.90,0.00),v40,z0,tPen\WObj:=wPaper;
    MoveL Offs(pOrigin,219.10,259.04,0.00),v40,z0,tPen\WObj:=wPaper;
    MoveL Offs(pOrigin,218.05,258.60,0.00),v40,z0,tPen\WObj:=wPaper;
    MoveL Offs(pOrigin,215.64,261.00,0.00),v40,z0,tPen\WObj:=wPaper;
    MoveL Offs(pOrigin,214.75,260.41,0.00),v40,z0,tPen\WObj:=wPaper;
    MoveL Offs(pOrigin,217.00,258.15,0.00),v40,z0,tPen\WObj:=wPaper;
    MoveL Offs(pOrigin,216.76,258.87,0.00),v40,z0,tPen\WObj:=wPaper;
    MoveL Offs(pOrigin,223.53,265.63,0.00),v40,fine,tPen\WObj:=wPaper;
    MoveL Offs(pOrigin,223.53,265.63,6.00),v60,z5,tPen\WObj:=wPaper;
    MoveL Offs(pOrigin,223.23,266.83,6.00),vTravel,z5,tPen\WObj:=wPaper;
    MoveL Offs(pOrigin,223.23,266.83,0.00),v60,z0,tPen\WObj:=wPaper;
    MoveL Offs(pOrigin,228.64,272.24,0.00),v40,z0,tPen\WObj:=wPaper;
    MoveL Offs(pOrigin,228.04,272.50,0.00),v40,z0,tPen\WObj:=wPaper;
    MoveL Offs(pOrigin,239.01,261.53,0.00),v40,z0,tPen\WObj:=wPaper;
    MoveL Offs(pOrigin,238.19,260.89,0.00),v40,z0,tPen\WObj:=wPaper;
    MoveL Offs(pOrigin,235.19,257.88,0.00),v40,z0,tPen\WObj:=wPaper;
    MoveL Offs(pOrigin,234.59,258.78,0.00),v40,z0,tPen\WObj:=wPaper;
    MoveL Offs(pOrigin,238.50,262.68,0.00),v40,z0,tPen\WObj:=wPaper;
    MoveL Offs(pOrigin,239.01,263.03,0.00),v40,z0,tPen\WObj:=wPaper;
    MoveL Offs(pOrigin,229.54,272.49,0.00),v40,z0,tPen\WObj:=wPaper;
    MoveL Offs(pOrigin,229.84,271.95,0.00),v40,z0,tPen\WObj:=wPaper;
    MoveL Offs(pOrigin,224.73,266.84,0.00),v40,fine,tPen\WObj:=wPaper;
    MoveL Offs(pOrigin,224.73,266.84,6.00),v60,z5,tPen\WObj:=wPaper;
    MoveL Offs(pOrigin,224.50,268.44,6.00),vTravel,z5,tPen\WObj:=wPaper;
    MoveL Offs(pOrigin,224.50,268.44,0.00),v60,z0,tPen\WObj:=wPaper;
    MoveL Offs(pOrigin,222.38,268.44,0.00),v40,z0,tPen\WObj:=wPaper;
    MoveL Offs(pOrigin,222.38,268.92,0.00),v40,z0,tPen\WObj:=wPaper;
    MoveL Offs(pOrigin,219.19,268.50,0.00),v40,z0,tPen\WObj:=wPaper;
    MoveL Offs(pOrigin,219.19,268.50,0.00),v40,z0,tPen\WObj:=wPaper;
    MoveL Offs(pOrigin,215.15,268.08,0.00),v40,z0,tPen\WObj:=wPaper;
    MoveL Offs(pOrigin,215.15,268.71,0.00),v40,z0,tPen\WObj:=wPaper;
    MoveL Offs(pOrigin,214.73,267.65,0.00),v40,z0,tPen\WObj:=wPaper;
    MoveL Offs(pOrigin,213.88,267.86,0.00),v40,z0,tPen\WObj:=wPaper;
    MoveL Offs(pOrigin,213.88,267.86,0.00),v40,z0,tPen\WObj:=wPaper;
    MoveL Offs(pOrigin,209.41,266.30,0.00),v40,z0,tPen\WObj:=wPaper;
    MoveL Offs(pOrigin,208.77,265.17,0.00),v40,z0,tPen\WObj:=wPaper;
    MoveL Offs(pOrigin,207.57,264.67,0.00),v40,z0,tPen\WObj:=wPaper;
    MoveL Offs(pOrigin,207.29,263.61,0.00),v40,z0,tPen\WObj:=wPaper;
    MoveL Offs(pOrigin,207.29,263.61,0.00),v40,z0,tPen\WObj:=wPaper;
    MoveL Offs(pOrigin,204.52,263.12,0.00),v40,z0,tPen\WObj:=wPaper;
    MoveL Offs(pOrigin,204.10,261.91,0.00),v40,z0,tPen\WObj:=wPaper;
    MoveL Offs(pOrigin,204.10,261.91,0.00),v40,z0,tPen\WObj:=wPaper;
    MoveL Offs(pOrigin,207.07,260.92,0.00),v40,z0,tPen\WObj:=wPaper;
    MoveL Offs(pOrigin,207.29,263.61,0.00),v40,z0,tPen\WObj:=wPaper;
    MoveL Offs(pOrigin,207.08,264.22,0.00),v40,z0,tPen\WObj:=wPaper;
    MoveL Offs(pOrigin,198.79,264.22,0.00),v40,z0,tPen\WObj:=wPaper;
    MoveL Offs(pOrigin,199.60,264.04,0.00),v40,z0,tPen\WObj:=wPaper;
    MoveL Offs(pOrigin,199.60,270.62,0.00),v40,z0,tPen\WObj:=wPaper;
    MoveL Offs(pOrigin,199.00,270.41,0.00),v40,z0,tPen\WObj:=wPaper;
    MoveL Offs(pOrigin,200.91,274.45,0.00),v40,z0,tPen\WObj:=wPaper;
    MoveL Offs(pOrigin,200.65,274.24,0.00),v40,z0,tPen\WObj:=wPaper;
    MoveL Offs(pOrigin,200.65,275.51,0.00),v40,z0,tPen\WObj:=wPaper;
    MoveL Offs(pOrigin,201.71,275.09,0.00),v40,z0,tPen\WObj:=wPaper;
    MoveL Offs(pOrigin,201.71,276.79,0.00),v40,z0,tPen\WObj:=wPaper;
    MoveL Offs(pOrigin,202.77,276.36,0.00),v40,z0,tPen\WObj:=wPaper;
    MoveL Offs(pOrigin,202.77,278.27,0.00),v40,z0,tPen\WObj:=wPaper;
    MoveL Offs(pOrigin,203.68,277.94,0.00),v40,z0,tPen\WObj:=wPaper;
    MoveL Offs(pOrigin,201.76,277.94,0.00),v40,fine,tPen\WObj:=wPaper;
    MoveL Offs(pOrigin,201.76,277.94,6.00),v60,z5,tPen\WObj:=wPaper;
    MoveL Offs(pOrigin,200.06,276.79,6.00),vTravel,z5,tPen\WObj:=wPaper;
    MoveL Offs(pOrigin,200.06,276.79,0.00),v60,z0,tPen\WObj:=wPaper;
    MoveL Offs(pOrigin,200.49,277.21,0.00),v40,z0,tPen\WObj:=wPaper;
    MoveL Offs(pOrigin,200.06,276.79,0.00),v40,z0,tPen\WObj:=wPaper;
    MoveL Offs(pOrigin,199.64,276.89,0.00),v40,z0,tPen\WObj:=wPaper;
    MoveL Offs(pOrigin,193.48,276.89,0.00),v40,z0,tPen\WObj:=wPaper;
    MoveL Offs(pOrigin,193.00,276.93,0.00),v40,z0,tPen\WObj:=wPaper;
    MoveL Offs(pOrigin,205.77,289.70,0.00),v40,z0,tPen\WObj:=wPaper;
    MoveL Offs(pOrigin,205.80,289.54,0.00),v40,z0,tPen\WObj:=wPaper;
    MoveL Offs(pOrigin,206.23,289.75,0.00),v40,z0,tPen\WObj:=wPaper;
    MoveL Offs(pOrigin,205.80,289.54,0.00),v40,fine,tPen\WObj:=wPaper;
    MoveL Offs(pOrigin,205.80,289.54,6.00),v60,z5,tPen\WObj:=wPaper;
    MoveL Offs(pOrigin,205.16,290.62,6.00),vTravel,z5,tPen\WObj:=wPaper;
    MoveL Offs(pOrigin,205.16,290.62,0.00),v60,z0,tPen\WObj:=wPaper;
    MoveL Offs(pOrigin,201.55,290.62,0.00),v40,fine,tPen\WObj:=wPaper;
    MoveL Offs(pOrigin,201.55,290.62,6.00),v60,z5,tPen\WObj:=wPaper;
    MoveL Offs(pOrigin,200.27,291.66,6.00),vTravel,z5,tPen\WObj:=wPaper;
    MoveL Offs(pOrigin,200.27,291.66,0.00),v60,z0,tPen\WObj:=wPaper;
    MoveL Offs(pOrigin,200.70,291.02,0.00),v40,z0,tPen\WObj:=wPaper;
    MoveL Offs(pOrigin,200.13,289.54,0.00),v40,z0,tPen\WObj:=wPaper;
    MoveL Offs(pOrigin,198.15,286.56,0.00),v40,z0,tPen\WObj:=wPaper;
    MoveL Offs(pOrigin,197.30,286.14,0.00),v40,fine,tPen\WObj:=wPaper;
    MoveL Offs(pOrigin,197.30,286.14,6.00),v60,z5,tPen\WObj:=wPaper;
    MoveL Offs(pOrigin,197.94,284.44,6.00),vTravel,z5,tPen\WObj:=wPaper;
    MoveL Offs(pOrigin,197.94,284.44,0.00),v60,z0,tPen\WObj:=wPaper;
    MoveL Offs(pOrigin,197.80,283.80,0.00),v40,z0,tPen\WObj:=wPaper;
    MoveL Offs(pOrigin,196.88,282.74,0.00),v40,z0,tPen\WObj:=wPaper;
    MoveL Offs(pOrigin,196.02,282.45,0.00),v40,z0,tPen\WObj:=wPaper;
    MoveL Offs(pOrigin,194.32,281.04,0.00),v40,z0,tPen\WObj:=wPaper;
    MoveL Offs(pOrigin,195.37,280.82,0.00),v40,z0,tPen\WObj:=wPaper;
    MoveL Offs(pOrigin,195.37,274.66,0.00),v40,z0,tPen\WObj:=wPaper;
    MoveL Offs(pOrigin,194.75,274.78,0.00),v40,z0,tPen\WObj:=wPaper;
    MoveL Offs(pOrigin,204.52,274.78,0.00),v40,z0,tPen\WObj:=wPaper;
    MoveL Offs(pOrigin,203.82,274.24,0.00),v40,z0,tPen\WObj:=wPaper;
    MoveL Offs(pOrigin,203.82,263.19,0.00),v40,z0,tPen\WObj:=wPaper;
    MoveL Offs(pOrigin,203.89,262.10,0.00),v40,z0,tPen\WObj:=wPaper;
    MoveL Offs(pOrigin,202.19,262.10,0.00),v40,z0,tPen\WObj:=wPaper;
    MoveL Offs(pOrigin,201.98,261.91,0.00),v40,z0,tPen\WObj:=wPaper;
    MoveL Offs(pOrigin,201.69,260.00,0.00),v40,z0,tPen\WObj:=wPaper;
    MoveL Offs(pOrigin,200.91,259.79,0.00),v40,z0,tPen\WObj:=wPaper;
    MoveL Offs(pOrigin,200.84,259.79,0.00),v40,z0,tPen\WObj:=wPaper;
    MoveL Offs(pOrigin,200.63,260.35,0.00),v40,z0,tPen\WObj:=wPaper;
    MoveL Offs(pOrigin,199.85,260.64,0.00),v40,z0,tPen\WObj:=wPaper;
    MoveL Offs(pOrigin,199.00,260.50,0.00),v40,z0,tPen\WObj:=wPaper;
    MoveL Offs(pOrigin,198.57,260.00,0.00),v40,z0,tPen\WObj:=wPaper;
    MoveL Offs(pOrigin,198.79,259.22,0.00),v40,z0,tPen\WObj:=wPaper;
    MoveL Offs(pOrigin,200.84,259.79,0.00),v40,z0,tPen\WObj:=wPaper;
    MoveL Offs(pOrigin,200.29,260.32,0.00),v40,z0,tPen\WObj:=wPaper;
    MoveL Offs(pOrigin,198.64,258.67,0.00),v40,z0,tPen\WObj:=wPaper;
    MoveL Offs(pOrigin,198.57,259.15,0.00),v40,z0,tPen\WObj:=wPaper;
    MoveL Offs(pOrigin,198.15,257.24,0.00),v40,z0,tPen\WObj:=wPaper;
    MoveL Offs(pOrigin,198.36,253.84,0.00),v40,z0,tPen\WObj:=wPaper;
    MoveL Offs(pOrigin,199.99,250.23,0.00),v40,z0,tPen\WObj:=wPaper;
    MoveL Offs(pOrigin,201.12,249.59,0.00),v40,z0,tPen\WObj:=wPaper;
    MoveL Offs(pOrigin,201.12,249.59,0.00),v40,z0,tPen\WObj:=wPaper;
    MoveL Offs(pOrigin,202.97,243.85,0.00),v40,z0,tPen\WObj:=wPaper;
    MoveL Offs(pOrigin,205.80,238.32,0.00),v40,z0,tPen\WObj:=wPaper;
    MoveL Offs(pOrigin,206.42,238.86,0.00),v40,z0,tPen\WObj:=wPaper;
    MoveL Offs(pOrigin,195.76,249.53,0.00),v40,z0,tPen\WObj:=wPaper;
    MoveL Offs(pOrigin,196.24,249.80,0.00),v40,z0,tPen\WObj:=wPaper;
  ENDPROC

  PROC DrawPart112()
    MoveL Offs(pOrigin,196.02,250.23,0.00),v40,z0,tPen\WObj:=wPaper;
    MoveL Offs(pOrigin,196.24,249.80,0.00),v40,z0,tPen\WObj:=wPaper;
    MoveL Offs(pOrigin,196.07,250.12,0.00),v40,z0,tPen\WObj:=wPaper;
    MoveL Offs(pOrigin,197.42,251.47,0.00),v40,z0,tPen\WObj:=wPaper;
    MoveL Offs(pOrigin,197.30,250.86,0.00),v40,z0,tPen\WObj:=wPaper;
    MoveL Offs(pOrigin,197.09,251.29,0.00),v40,z0,tPen\WObj:=wPaper;
    MoveL Offs(pOrigin,197.30,250.86,0.00),v40,z0,tPen\WObj:=wPaper;
    MoveL Offs(pOrigin,197.86,250.43,0.00),v40,z0,tPen\WObj:=wPaper;
    MoveL Offs(pOrigin,196.66,249.22,0.00),v40,z0,tPen\WObj:=wPaper;
    MoveL Offs(pOrigin,197.26,248.33,0.00),v40,z0,tPen\WObj:=wPaper;
    MoveL Offs(pOrigin,198.61,249.68,0.00),v40,z0,tPen\WObj:=wPaper;
    MoveL Offs(pOrigin,198.57,248.74,0.00),v40,z0,tPen\WObj:=wPaper;
    MoveL Offs(pOrigin,198.15,249.38,0.00),v40,z0,tPen\WObj:=wPaper;
    MoveL Offs(pOrigin,198.57,248.74,0.00),v40,z0,tPen\WObj:=wPaper;
    MoveL Offs(pOrigin,199.06,248.63,0.00),v40,z0,tPen\WObj:=wPaper;
    MoveL Offs(pOrigin,197.85,247.43,0.00),v40,z0,tPen\WObj:=wPaper;
    MoveL Offs(pOrigin,197.73,247.68,0.00),v40,z0,tPen\WObj:=wPaper;
    MoveL Offs(pOrigin,197.30,248.31,0.00),v40,z0,tPen\WObj:=wPaper;
    MoveL Offs(pOrigin,197.73,247.68,0.00),v40,fine,tPen\WObj:=wPaper;
    MoveL Offs(pOrigin,197.73,247.68,6.00),v60,z5,tPen\WObj:=wPaper;
    MoveL Offs(pOrigin,198.30,246.38,6.00),vTravel,z5,tPen\WObj:=wPaper;
    MoveL Offs(pOrigin,198.30,246.38,0.00),v60,z0,tPen\WObj:=wPaper;
    MoveL Offs(pOrigin,199.65,247.74,0.00),v40,z0,tPen\WObj:=wPaper;
    MoveL Offs(pOrigin,199.64,247.04,0.00),v40,z0,tPen\WObj:=wPaper;
    MoveL Offs(pOrigin,199.43,247.46,0.00),v40,z0,tPen\WObj:=wPaper;
    MoveL Offs(pOrigin,199.64,247.04,0.00),v40,z0,tPen\WObj:=wPaper;
    MoveL Offs(pOrigin,200.25,246.84,0.00),v40,z0,tPen\WObj:=wPaper;
    MoveL Offs(pOrigin,198.90,245.49,0.00),v40,z0,tPen\WObj:=wPaper;
    MoveL Offs(pOrigin,198.79,245.98,0.00),v40,z0,tPen\WObj:=wPaper;
    MoveL Offs(pOrigin,198.36,246.61,0.00),v40,z0,tPen\WObj:=wPaper;
    MoveL Offs(pOrigin,198.79,245.98,0.00),v40,fine,tPen\WObj:=wPaper;
    MoveL Offs(pOrigin,198.79,245.98,6.00),v60,z5,tPen\WObj:=wPaper;
    MoveL Offs(pOrigin,197.56,246.23,6.00),vTravel,z5,tPen\WObj:=wPaper;
    MoveL Offs(pOrigin,197.56,246.23,0.00),v60,z0,tPen\WObj:=wPaper;
    MoveL Offs(pOrigin,204.78,239.02,0.00),v40,z0,tPen\WObj:=wPaper;
    MoveL Offs(pOrigin,203.73,238.57,0.00),v40,z0,tPen\WObj:=wPaper;
    MoveL Offs(pOrigin,199.07,243.23,0.00),v40,z0,tPen\WObj:=wPaper;
    MoveL Offs(pOrigin,199.79,243.39,0.00),v40,z0,tPen\WObj:=wPaper;
    MoveL Offs(pOrigin,201.29,244.89,0.00),v40,z0,tPen\WObj:=wPaper;
    MoveL Offs(pOrigin,201.74,243.85,0.00),v40,z0,tPen\WObj:=wPaper;
    MoveL Offs(pOrigin,200.24,242.34,0.00),v40,z0,tPen\WObj:=wPaper;
    MoveL Offs(pOrigin,200.70,242.04,0.00),v40,z0,tPen\WObj:=wPaper;
    MoveL Offs(pOrigin,201.76,242.04,0.00),v40,z0,tPen\WObj:=wPaper;
    MoveL Offs(pOrigin,202.18,242.80,0.00),v40,z0,tPen\WObj:=wPaper;
    MoveL Offs(pOrigin,197.08,237.69,0.00),v40,z0,tPen\WObj:=wPaper;
    MoveL Offs(pOrigin,197.59,237.24,0.00),v40,z0,tPen\WObj:=wPaper;
    MoveL Offs(pOrigin,194.89,239.94,0.00),v40,z0,tPen\WObj:=wPaper;
    MoveL Offs(pOrigin,194.38,239.48,0.00),v40,z0,tPen\WObj:=wPaper;
    MoveL Offs(pOrigin,191.68,236.78,0.00),v40,z0,tPen\WObj:=wPaper;
    MoveL Offs(pOrigin,191.30,236.06,0.00),v40,z0,tPen\WObj:=wPaper;
    MoveL Offs(pOrigin,188.75,238.62,0.00),v40,z0,tPen\WObj:=wPaper;
    MoveL Offs(pOrigin,188.84,238.41,0.00),v40,z0,tPen\WObj:=wPaper;
    MoveL Offs(pOrigin,185.68,235.26,0.00),v40,z0,tPen\WObj:=wPaper;
    MoveL Offs(pOrigin,185.19,235.70,0.00),v40,z0,tPen\WObj:=wPaper;
    MoveL Offs(pOrigin,180.30,235.70,0.00),v40,z0,tPen\WObj:=wPaper;
    MoveL Offs(pOrigin,180.37,236.54,0.00),v40,z0,tPen\WObj:=wPaper;
    MoveL Offs(pOrigin,183.97,232.94,0.00),v40,z0,tPen\WObj:=wPaper;
    MoveL Offs(pOrigin,183.70,233.86,0.00),v40,z0,tPen\WObj:=wPaper;
    MoveL Offs(pOrigin,183.27,233.30,0.00),v40,z0,tPen\WObj:=wPaper;
    MoveL Offs(pOrigin,179.88,232.02,0.00),v40,z0,tPen\WObj:=wPaper;
    MoveL Offs(pOrigin,175.62,229.61,0.00),v40,z0,tPen\WObj:=wPaper;
    MoveL Offs(pOrigin,173.29,227.27,0.00),v40,z0,tPen\WObj:=wPaper;
    MoveL Offs(pOrigin,172.15,225.57,0.00),v40,z0,tPen\WObj:=wPaper;
    MoveL Offs(pOrigin,170.52,221.54,0.00),v40,z0,tPen\WObj:=wPaper;
    MoveL Offs(pOrigin,169.68,217.50,0.00),v40,z0,tPen\WObj:=wPaper;
    MoveL Offs(pOrigin,169.68,210.49,0.00),v40,z0,tPen\WObj:=wPaper;
    MoveL Offs(pOrigin,170.74,204.32,0.00),v40,z0,tPen\WObj:=wPaper;
    MoveL Offs(pOrigin,172.72,198.02,0.00),v40,z0,tPen\WObj:=wPaper;
    MoveL Offs(pOrigin,174.35,198.30,0.00),v40,z0,tPen\WObj:=wPaper;
    MoveL Offs(pOrigin,181.57,201.28,0.00),v40,z0,tPen\WObj:=wPaper;
    MoveL Offs(pOrigin,197.30,209.28,0.00),v40,z0,tPen\WObj:=wPaper;
    MoveL Offs(pOrigin,201.98,211.20,0.00),v40,z0,tPen\WObj:=wPaper;
    MoveL Offs(pOrigin,207.29,212.61,0.00),v40,z0,tPen\WObj:=wPaper;
    MoveL Offs(pOrigin,216.00,213.89,0.00),v40,z0,tPen\WObj:=wPaper;
    MoveL Offs(pOrigin,215.79,214.74,0.00),v40,z0,tPen\WObj:=wPaper;
    MoveL Offs(pOrigin,211.47,219.84,0.00),v40,z0,tPen\WObj:=wPaper;
    MoveL Offs(pOrigin,209.34,223.66,0.00),v40,z0,tPen\WObj:=wPaper;
    MoveL Offs(pOrigin,208.07,226.85,0.00),v40,z0,tPen\WObj:=wPaper;
    MoveL Offs(pOrigin,206.65,226.85,0.00),v40,z0,tPen\WObj:=wPaper;
    MoveL Offs(pOrigin,204.52,227.91,0.00),v40,z0,tPen\WObj:=wPaper;
    MoveL Offs(pOrigin,202.97,230.04,0.00),v40,z0,tPen\WObj:=wPaper;
    MoveL Offs(pOrigin,202.19,232.66,0.00),v40,z0,tPen\WObj:=wPaper;
    MoveL Offs(pOrigin,200.49,232.59,0.00),v40,z0,tPen\WObj:=wPaper;
    MoveL Offs(pOrigin,194.96,231.31,0.00),v40,z0,tPen\WObj:=wPaper;
    MoveL Offs(pOrigin,189.23,229.47,0.00),v40,z0,tPen\WObj:=wPaper;
    MoveL Offs(pOrigin,184.55,227.42,0.00),v40,z0,tPen\WObj:=wPaper;
    MoveL Offs(pOrigin,183.49,227.27,0.00),v40,z0,tPen\WObj:=wPaper;
    MoveL Offs(pOrigin,183.49,227.27,0.00),v40,z0,tPen\WObj:=wPaper;
    MoveL Offs(pOrigin,183.49,226.64,0.00),v40,z0,tPen\WObj:=wPaper;
    MoveL Offs(pOrigin,182.43,226.64,0.00),v40,z0,tPen\WObj:=wPaper;
    MoveL Offs(pOrigin,182.43,226.64,0.00),v40,z0,tPen\WObj:=wPaper;
    MoveL Offs(pOrigin,182.85,227.49,0.00),v40,z0,tPen\WObj:=wPaper;
    MoveL Offs(pOrigin,183.49,227.70,0.00),v40,z0,tPen\WObj:=wPaper;
    MoveL Offs(pOrigin,183.49,227.70,0.00),v40,z0,tPen\WObj:=wPaper;
    MoveL Offs(pOrigin,186.25,229.26,0.00),v40,z0,tPen\WObj:=wPaper;
    MoveL Offs(pOrigin,190.93,231.17,0.00),v40,z0,tPen\WObj:=wPaper;
    MoveL Offs(pOrigin,196.45,232.80,0.00),v40,z0,tPen\WObj:=wPaper;
    MoveL Offs(pOrigin,201.98,233.93,0.00),v40,z0,tPen\WObj:=wPaper;
    MoveL Offs(pOrigin,202.19,235.56,0.00),v40,z0,tPen\WObj:=wPaper;
    MoveL Offs(pOrigin,201.69,238.32,0.00),v40,z0,tPen\WObj:=wPaper;
    MoveL Offs(pOrigin,201.34,238.61,0.00),v40,z0,tPen\WObj:=wPaper;
    MoveL Offs(pOrigin,199.85,238.54,0.00),v40,z0,tPen\WObj:=wPaper;
    MoveL Offs(pOrigin,187.10,236.20,0.00),v40,z0,tPen\WObj:=wPaper;
    MoveL Offs(pOrigin,179.88,234.29,0.00),v40,z0,tPen\WObj:=wPaper;
    MoveL Offs(pOrigin,174.77,232.45,0.00),v40,z0,tPen\WObj:=wPaper;
    MoveL Offs(pOrigin,171.38,230.75,0.00),v40,z0,tPen\WObj:=wPaper;
    MoveL Offs(pOrigin,170.10,229.19,0.00),v40,z0,tPen\WObj:=wPaper;
    MoveL Offs(pOrigin,170.10,229.19,0.00),v40,z0,tPen\WObj:=wPaper;
    MoveL Offs(pOrigin,169.82,227.91,0.00),v40,z0,tPen\WObj:=wPaper;
    MoveL Offs(pOrigin,168.40,225.79,0.00),v40,z0,tPen\WObj:=wPaper;
    MoveL Offs(pOrigin,168.40,225.79,0.00),v40,z0,tPen\WObj:=wPaper;
    MoveL Offs(pOrigin,167.48,225.36,0.00),v40,z0,tPen\WObj:=wPaper;
    MoveL Offs(pOrigin,165.78,221.54,0.00),v40,z0,tPen\WObj:=wPaper;
    MoveL Offs(pOrigin,164.79,217.71,0.00),v40,z0,tPen\WObj:=wPaper;
    MoveL Offs(pOrigin,164.36,214.10,0.00),v40,z0,tPen\WObj:=wPaper;
    MoveL Offs(pOrigin,164.36,209.21,0.00),v40,z0,tPen\WObj:=wPaper;
    MoveL Offs(pOrigin,164.79,204.96,0.00),v40,z0,tPen\WObj:=wPaper;
    MoveL Offs(pOrigin,166.70,196.04,0.00),v40,z0,tPen\WObj:=wPaper;
    MoveL Offs(pOrigin,166.27,195.47,0.00),v40,z0,tPen\WObj:=wPaper;
    MoveL Offs(pOrigin,161.60,194.12,0.00),v40,z0,tPen\WObj:=wPaper;
  ENDPROC

  PROC DrawPart113()
    MoveL Offs(pOrigin,161.18,194.55,0.00),v40,z0,tPen\WObj:=wPaper;
    MoveL Offs(pOrigin,161.18,208.15,0.00),v40,z0,tPen\WObj:=wPaper;
    MoveL Offs(pOrigin,161.60,213.89,0.00),v40,z0,tPen\WObj:=wPaper;
    MoveL Offs(pOrigin,162.24,217.50,0.00),v40,z0,tPen\WObj:=wPaper;
    MoveL Offs(pOrigin,163.23,220.90,0.00),v40,z0,tPen\WObj:=wPaper;
    MoveL Offs(pOrigin,165.43,224.94,0.00),v40,z0,tPen\WObj:=wPaper;
    MoveL Offs(pOrigin,168.82,228.76,0.00),v40,z0,tPen\WObj:=wPaper;
    MoveL Offs(pOrigin,170.10,229.19,0.00),v40,z0,tPen\WObj:=wPaper;
    MoveL Offs(pOrigin,169.46,229.37,0.00),v40,z0,tPen\WObj:=wPaper;
    MoveL Offs(pOrigin,167.55,229.37,0.00),v40,z0,tPen\WObj:=wPaper;
    MoveL Offs(pOrigin,167.20,230.29,0.00),v40,z0,tPen\WObj:=wPaper;
    MoveL Offs(pOrigin,172.61,224.88,0.00),v40,z0,tPen\WObj:=wPaper;
    MoveL Offs(pOrigin,171.80,224.51,0.00),v40,z0,tPen\WObj:=wPaper;
    MoveL Offs(pOrigin,172.01,224.94,0.00),v40,z0,tPen\WObj:=wPaper;
    MoveL Offs(pOrigin,171.80,224.51,0.00),v40,z0,tPen\WObj:=wPaper;
    MoveL Offs(pOrigin,171.72,224.28,0.00),v40,z0,tPen\WObj:=wPaper;
    MoveL Offs(pOrigin,168.26,220.83,0.00),v40,z0,tPen\WObj:=wPaper;
    MoveL Offs(pOrigin,169.04,220.92,0.00),v40,z0,tPen\WObj:=wPaper;
    MoveL Offs(pOrigin,170.10,220.92,0.00),v40,z0,tPen\WObj:=wPaper;
    MoveL Offs(pOrigin,170.83,220.69,0.00),v40,z0,tPen\WObj:=wPaper;
    MoveL Offs(pOrigin,164.37,227.16,0.00),v40,z0,tPen\WObj:=wPaper;
    MoveL Offs(pOrigin,164.36,226.43,0.00),v40,z0,tPen\WObj:=wPaper;
    MoveL Offs(pOrigin,165.21,227.49,0.00),v40,z0,tPen\WObj:=wPaper;
    MoveL Offs(pOrigin,164.36,226.43,0.00),v40,z0,tPen\WObj:=wPaper;
    MoveL Offs(pOrigin,164.79,226.20,0.00),v40,z0,tPen\WObj:=wPaper;
    MoveL Offs(pOrigin,166.06,226.20,0.00),v40,z0,tPen\WObj:=wPaper;
    MoveL Offs(pOrigin,166.06,226.00,0.00),v40,z0,tPen\WObj:=wPaper;
    MoveL Offs(pOrigin,166.49,226.43,0.00),v40,z0,tPen\WObj:=wPaper;
    MoveL Offs(pOrigin,166.06,226.00,0.00),v40,z0,tPen\WObj:=wPaper;
    MoveL Offs(pOrigin,166.93,225.46,0.00),v40,z0,tPen\WObj:=wPaper;
    MoveL Offs(pOrigin,168.73,227.27,0.00),v40,z0,tPen\WObj:=wPaper;
    MoveL Offs(pOrigin,168.19,228.31,0.00),v40,z0,tPen\WObj:=wPaper;
    MoveL Offs(pOrigin,166.49,228.31,0.00),v40,z0,tPen\WObj:=wPaper;
    MoveL Offs(pOrigin,166.49,228.98,0.00),v40,z0,tPen\WObj:=wPaper;
    MoveL Offs(pOrigin,166.91,229.40,0.00),v40,z0,tPen\WObj:=wPaper;
    MoveL Offs(pOrigin,166.49,228.98,0.00),v40,z0,tPen\WObj:=wPaper;
    MoveL Offs(pOrigin,166.46,229.55,0.00),v40,z0,tPen\WObj:=wPaper;
    MoveL Offs(pOrigin,172.17,223.84,0.00),v40,z0,tPen\WObj:=wPaper;
    MoveL Offs(pOrigin,171.38,224.09,0.00),v40,z0,tPen\WObj:=wPaper;
    MoveL Offs(pOrigin,170.10,224.09,0.00),v40,z0,tPen\WObj:=wPaper;
    MoveL Offs(pOrigin,169.32,224.87,0.00),v40,z0,tPen\WObj:=wPaper;
    MoveL Offs(pOrigin,181.04,236.59,0.00),v40,z0,tPen\WObj:=wPaper;
    MoveL Offs(pOrigin,181.41,236.99,0.00),v40,z0,tPen\WObj:=wPaper;
    MoveL Offs(pOrigin,185.02,233.38,0.00),v40,z0,tPen\WObj:=wPaper;
    MoveL Offs(pOrigin,185.92,233.98,0.00),v40,z0,tPen\WObj:=wPaper;
    MoveL Offs(pOrigin,182.61,237.29,0.00),v40,z0,tPen\WObj:=wPaper;
    MoveL Offs(pOrigin,183.14,237.20,0.00),v40,z0,tPen\WObj:=wPaper;
    MoveL Offs(pOrigin,168.72,222.77,0.00),v40,z0,tPen\WObj:=wPaper;
    MoveL Offs(pOrigin,169.25,221.98,0.00),v40,z0,tPen\WObj:=wPaper;
    MoveL Offs(pOrigin,170.52,221.98,0.00),v40,z0,tPen\WObj:=wPaper;
    MoveL Offs(pOrigin,170.96,222.03,0.00),v40,z0,tPen\WObj:=wPaper;
    MoveL Offs(pOrigin,168.11,219.18,0.00),v40,z0,tPen\WObj:=wPaper;
    MoveL Offs(pOrigin,168.82,219.86,0.00),v40,z0,tPen\WObj:=wPaper;
    MoveL Offs(pOrigin,169.89,219.86,0.00),v40,z0,tPen\WObj:=wPaper;
    MoveL Offs(pOrigin,170.36,219.93,0.00),v40,z0,tPen\WObj:=wPaper;
    MoveL Offs(pOrigin,167.95,217.53,0.00),v40,z0,tPen\WObj:=wPaper;
    MoveL Offs(pOrigin,168.40,216.70,0.00),v40,z0,tPen\WObj:=wPaper;
    MoveL Offs(pOrigin,169.46,216.70,0.00),v40,z0,tPen\WObj:=wPaper;
    MoveL Offs(pOrigin,169.90,216.49,0.00),v40,z0,tPen\WObj:=wPaper;
    MoveL Offs(pOrigin,167.64,214.23,0.00),v40,fine,tPen\WObj:=wPaper;
    MoveL Offs(pOrigin,167.64,214.23,6.00),v60,z5,tPen\WObj:=wPaper;
    MoveL Offs(pOrigin,166.30,214.38,6.00),vTravel,z5,tPen\WObj:=wPaper;
    MoveL Offs(pOrigin,166.30,214.38,0.00),v60,z0,tPen\WObj:=wPaper;
    MoveL Offs(pOrigin,164.34,212.42,0.00),v40,z0,tPen\WObj:=wPaper;
    MoveL Offs(pOrigin,163.66,212.93,0.00),v40,z0,tPen\WObj:=wPaper;
    MoveL Offs(pOrigin,166.67,209.92,0.00),v40,z0,tPen\WObj:=wPaper;
    MoveL Offs(pOrigin,166.13,209.73,0.00),v40,z0,tPen\WObj:=wPaper;
    MoveL Offs(pOrigin,164.33,207.93,0.00),v40,z0,tPen\WObj:=wPaper;
    MoveL Offs(pOrigin,163.68,208.43,0.00),v40,z0,tPen\WObj:=wPaper;
    MoveL Offs(pOrigin,167.13,204.98,0.00),v40,z0,tPen\WObj:=wPaper;
    MoveL Offs(pOrigin,166.71,204.34,0.00),v40,z0,tPen\WObj:=wPaper;
    MoveL Offs(pOrigin,164.91,202.54,0.00),v40,z0,tPen\WObj:=wPaper;
    MoveL Offs(pOrigin,164.45,201.69,0.00),v40,z0,tPen\WObj:=wPaper;
    MoveL Offs(pOrigin,173.16,192.97,0.00),v40,z0,tPen\WObj:=wPaper;
    MoveL Offs(pOrigin,172.11,192.53,0.00),v40,z0,tPen\WObj:=wPaper;
    MoveL Offs(pOrigin,164.90,199.74,0.00),v40,z0,tPen\WObj:=wPaper;
    MoveL Offs(pOrigin,165.35,199.99,0.00),v40,z0,tPen\WObj:=wPaper;
    MoveL Offs(pOrigin,167.16,201.80,0.00),v40,z0,tPen\WObj:=wPaper;
    MoveL Offs(pOrigin,167.74,201.38,0.00),v40,z0,tPen\WObj:=wPaper;
    MoveL Offs(pOrigin,163.99,205.14,0.00),v40,z0,tPen\WObj:=wPaper;
    MoveL Offs(pOrigin,164.47,205.08,0.00),v40,z0,tPen\WObj:=wPaper;
    MoveL Offs(pOrigin,166.27,206.89,0.00),v40,z0,tPen\WObj:=wPaper;
    MoveL Offs(pOrigin,166.83,206.78,0.00),v40,z0,tPen\WObj:=wPaper;
    MoveL Offs(pOrigin,163.67,209.93,0.00),v40,z0,tPen\WObj:=wPaper;
    MoveL Offs(pOrigin,164.04,210.63,0.00),v40,z0,tPen\WObj:=wPaper;
    MoveL Offs(pOrigin,166.14,212.73,0.00),v40,fine,tPen\WObj:=wPaper;
    MoveL Offs(pOrigin,166.14,212.73,6.00),v60,z5,tPen\WObj:=wPaper;
    MoveL Offs(pOrigin,167.64,212.73,6.00),vTravel,z5,tPen\WObj:=wPaper;
    MoveL Offs(pOrigin,167.64,212.73,0.00),v60,z0,tPen\WObj:=wPaper;
    MoveL Offs(pOrigin,169.89,214.99,0.00),v40,z0,tPen\WObj:=wPaper;
    MoveL Offs(pOrigin,170.25,215.30,0.00),v40,z0,tPen\WObj:=wPaper;
    MoveL Offs(pOrigin,161.98,223.57,0.00),v40,z0,tPen\WObj:=wPaper;
    MoveL Offs(pOrigin,162.24,222.81,0.00),v40,z0,tPen\WObj:=wPaper;
    MoveL Offs(pOrigin,162.45,223.24,0.00),v40,z0,tPen\WObj:=wPaper;
    MoveL Offs(pOrigin,162.24,222.81,0.00),v40,z0,tPen\WObj:=wPaper;
    MoveL Offs(pOrigin,162.88,223.03,0.00),v40,z0,tPen\WObj:=wPaper;
    MoveL Offs(pOrigin,163.94,223.03,0.00),v40,z0,tPen\WObj:=wPaper;
    MoveL Offs(pOrigin,164.15,223.02,0.00),v40,z0,tPen\WObj:=wPaper;
    MoveL Offs(pOrigin,164.36,223.45,0.00),v40,z0,tPen\WObj:=wPaper;
    MoveL Offs(pOrigin,164.15,223.02,0.00),v40,z0,tPen\WObj:=wPaper;
    MoveL Offs(pOrigin,164.52,223.06,0.00),v40,z0,tPen\WObj:=wPaper;
    MoveL Offs(pOrigin,160.62,219.15,0.00),v40,z0,tPen\WObj:=wPaper;
    MoveL Offs(pOrigin,160.35,219.23,0.00),v40,z0,tPen\WObj:=wPaper;
    MoveL Offs(pOrigin,162.75,216.82,0.00),v40,z0,tPen\WObj:=wPaper;
    MoveL Offs(pOrigin,162.11,216.16,0.00),v40,z0,tPen\WObj:=wPaper;
    MoveL Offs(pOrigin,159.70,213.76,0.00),v40,z0,tPen\WObj:=wPaper;
    MoveL Offs(pOrigin,159.31,214.29,0.00),v40,z0,tPen\WObj:=wPaper;
    MoveL Offs(pOrigin,162.02,211.58,0.00),v40,z0,tPen\WObj:=wPaper;
    MoveL Offs(pOrigin,161.64,211.22,0.00),v40,z0,tPen\WObj:=wPaper;
    MoveL Offs(pOrigin,159.69,209.26,0.00),v40,z0,tPen\WObj:=wPaper;
    MoveL Offs(pOrigin,159.18,209.94,0.00),v40,z0,tPen\WObj:=wPaper;
    MoveL Offs(pOrigin,161.73,207.39,0.00),v40,z0,tPen\WObj:=wPaper;
    MoveL Offs(pOrigin,161.33,207.92,0.00),v40,z0,tPen\WObj:=wPaper;
    MoveL Offs(pOrigin,159.38,205.97,0.00),v40,z0,tPen\WObj:=wPaper;
    MoveL Offs(pOrigin,159.04,205.60,0.00),v40,z0,tPen\WObj:=wPaper;
    MoveL Offs(pOrigin,161.74,202.90,0.00),v40,z0,tPen\WObj:=wPaper;
    MoveL Offs(pOrigin,161.32,203.43,0.00),v40,z0,tPen\WObj:=wPaper;
    MoveL Offs(pOrigin,159.37,201.47,0.00),v40,z0,tPen\WObj:=wPaper;
    MoveL Offs(pOrigin,158.75,201.41,0.00),v40,z0,tPen\WObj:=wPaper;
    MoveL Offs(pOrigin,161.76,198.40,0.00),v40,z0,tPen\WObj:=wPaper;
  ENDPROC

  PROC DrawPart114()
    MoveL Offs(pOrigin,161.30,198.93,0.00),v40,z0,tPen\WObj:=wPaper;
    MoveL Offs(pOrigin,159.20,196.83,0.00),v40,z0,tPen\WObj:=wPaper;
    MoveL Offs(pOrigin,158.77,196.91,0.00),v40,z0,tPen\WObj:=wPaper;
    MoveL Offs(pOrigin,165.08,190.60,0.00),v40,z0,tPen\WObj:=wPaper;
    MoveL Offs(pOrigin,166.13,191.05,0.00),v40,z0,tPen\WObj:=wPaper;
    MoveL Offs(pOrigin,158.76,198.41,0.00),v40,z0,tPen\WObj:=wPaper;
    MoveL Offs(pOrigin,159.21,198.33,0.00),v40,z0,tPen\WObj:=wPaper;
    MoveL Offs(pOrigin,161.31,200.43,0.00),v40,z0,tPen\WObj:=wPaper;
    MoveL Offs(pOrigin,161.75,199.90,0.00),v40,z0,tPen\WObj:=wPaper;
    MoveL Offs(pOrigin,158.75,202.91,0.00),v40,z0,tPen\WObj:=wPaper;
    MoveL Offs(pOrigin,159.37,202.97,0.00),v40,z0,tPen\WObj:=wPaper;
    MoveL Offs(pOrigin,161.32,204.93,0.00),v40,z0,tPen\WObj:=wPaper;
    MoveL Offs(pOrigin,161.74,204.39,0.00),v40,z0,tPen\WObj:=wPaper;
    MoveL Offs(pOrigin,159.04,207.10,0.00),v40,z0,tPen\WObj:=wPaper;
    MoveL Offs(pOrigin,159.38,207.47,0.00),v40,z0,tPen\WObj:=wPaper;
    MoveL Offs(pOrigin,161.64,209.72,0.00),v40,z0,tPen\WObj:=wPaper;
    MoveL Offs(pOrigin,162.02,210.09,0.00),v40,z0,tPen\WObj:=wPaper;
    MoveL Offs(pOrigin,159.32,212.79,0.00),v40,z0,tPen\WObj:=wPaper;
    MoveL Offs(pOrigin,159.55,212.11,0.00),v40,z0,tPen\WObj:=wPaper;
    MoveL Offs(pOrigin,161.65,214.21,0.00),v40,z0,tPen\WObj:=wPaper;
    MoveL Offs(pOrigin,162.46,214.13,0.00),v40,z0,tPen\WObj:=wPaper;
    MoveL Offs(pOrigin,159.75,216.83,0.00),v40,z0,tPen\WObj:=wPaper;
    MoveL Offs(pOrigin,160.16,217.21,0.00),v40,z0,tPen\WObj:=wPaper;
    MoveL Offs(pOrigin,163.17,220.21,0.00),v40,z0,tPen\WObj:=wPaper;
    MoveL Offs(pOrigin,162.66,219.86,0.00),v40,z0,tPen\WObj:=wPaper;
    MoveL Offs(pOrigin,161.60,219.86,0.00),v40,z0,tPen\WObj:=wPaper;
    MoveL Offs(pOrigin,160.64,220.43,0.00),v40,z0,tPen\WObj:=wPaper;
    MoveL Offs(pOrigin,163.05,218.02,0.00),v40,z0,tPen\WObj:=wPaper;
    MoveL Offs(pOrigin,162.56,218.11,0.00),v40,z0,tPen\WObj:=wPaper;
    MoveL Offs(pOrigin,160.01,215.56,0.00),v40,z0,tPen\WObj:=wPaper;
    MoveL Offs(pOrigin,159.61,215.49,0.00),v40,z0,tPen\WObj:=wPaper;
    MoveL Offs(pOrigin,162.16,212.93,0.00),v40,z0,tPen\WObj:=wPaper;
    MoveL Offs(pOrigin,161.80,212.87,0.00),v40,z0,tPen\WObj:=wPaper;
    MoveL Offs(pOrigin,159.69,210.76,0.00),v40,z0,tPen\WObj:=wPaper;
    MoveL Offs(pOrigin,159.17,211.44,0.00),v40,z0,tPen\WObj:=wPaper;
    MoveL Offs(pOrigin,162.03,208.59,0.00),v40,fine,tPen\WObj:=wPaper;
    MoveL Offs(pOrigin,162.03,208.59,6.00),v60,z5,tPen\WObj:=wPaper;
    MoveL Offs(pOrigin,161.33,206.42,6.00),vTravel,z5,tPen\WObj:=wPaper;
    MoveL Offs(pOrigin,161.33,206.42,0.00),v60,z0,tPen\WObj:=wPaper;
    MoveL Offs(pOrigin,159.37,204.47,0.00),v40,z0,tPen\WObj:=wPaper;
    MoveL Offs(pOrigin,158.74,204.40,0.00),v40,z0,tPen\WObj:=wPaper;
    MoveL Offs(pOrigin,161.75,201.40,0.00),v40,z0,tPen\WObj:=wPaper;
    MoveL Offs(pOrigin,161.31,201.93,0.00),v40,z0,tPen\WObj:=wPaper;
    MoveL Offs(pOrigin,159.21,199.83,0.00),v40,z0,tPen\WObj:=wPaper;
    MoveL Offs(pOrigin,158.76,199.91,0.00),v40,z0,tPen\WObj:=wPaper;
    MoveL Offs(pOrigin,161.76,196.90,0.00),v40,z0,tPen\WObj:=wPaper;
    MoveL Offs(pOrigin,161.30,197.44,0.00),v40,z0,tPen\WObj:=wPaper;
    MoveL Offs(pOrigin,159.20,195.33,0.00),v40,z0,tPen\WObj:=wPaper;
    MoveL Offs(pOrigin,158.77,195.42,0.00),v40,z0,tPen\WObj:=wPaper;
    MoveL Offs(pOrigin,163.73,190.46,0.00),v40,fine,tPen\WObj:=wPaper;
    MoveL Offs(pOrigin,163.73,190.46,6.00),v60,z5,tPen\WObj:=wPaper;
    MoveL Offs(pOrigin,162.38,190.31,6.00),vTravel,z5,tPen\WObj:=wPaper;
    MoveL Offs(pOrigin,162.38,190.31,0.00),v60,z0,tPen\WObj:=wPaper;
    MoveL Offs(pOrigin,158.63,194.07,0.00),v40,z0,tPen\WObj:=wPaper;
    MoveL Offs(pOrigin,159.48,193.46,0.00),v40,z0,tPen\WObj:=wPaper;
    MoveL Offs(pOrigin,164.58,193.46,0.00),v40,z0,tPen\WObj:=wPaper;
    MoveL Offs(pOrigin,163.98,192.65,0.00),v40,z0,tPen\WObj:=wPaper;
    MoveL Offs(pOrigin,168.49,197.16,0.00),v40,z0,tPen\WObj:=wPaper;
    MoveL Offs(pOrigin,168.19,196.63,0.00),v40,z0,tPen\WObj:=wPaper;
    MoveL Offs(pOrigin,166.70,196.63,0.00),v40,z0,tPen\WObj:=wPaper;
    MoveL Offs(pOrigin,166.86,195.82,0.00),v40,z0,tPen\WObj:=wPaper;
    MoveL Offs(pOrigin,166.86,194.76,0.00),v40,z0,tPen\WObj:=wPaper;
    MoveL Offs(pOrigin,166.28,195.58,0.00),v40,z0,tPen\WObj:=wPaper;
    MoveL Offs(pOrigin,171.16,195.58,0.00),v40,z0,tPen\WObj:=wPaper;
    MoveL Offs(pOrigin,170.88,195.07,0.00),v40,z0,tPen\WObj:=wPaper;
    MoveL Offs(pOrigin,174.79,198.97,0.00),v40,z0,tPen\WObj:=wPaper;
    MoveL Offs(pOrigin,174.49,199.11,0.00),v40,z0,tPen\WObj:=wPaper;
    MoveL Offs(pOrigin,178.70,194.90,0.00),v40,z0,tPen\WObj:=wPaper;
    MoveL Offs(pOrigin,179.12,195.84,0.00),v40,z0,tPen\WObj:=wPaper;
    MoveL Offs(pOrigin,180.32,197.04,0.00),v40,fine,tPen\WObj:=wPaper;
    MoveL Offs(pOrigin,180.32,197.04,6.00),v60,z5,tPen\WObj:=wPaper;
    MoveL Offs(pOrigin,181.52,196.75,6.00),vTravel,z5,tPen\WObj:=wPaper;
    MoveL Offs(pOrigin,181.52,196.75,0.00),v60,z0,tPen\WObj:=wPaper;
    MoveL Offs(pOrigin,183.77,199.00,0.00),v40,fine,tPen\WObj:=wPaper;
    MoveL Offs(pOrigin,183.77,199.00,6.00),v60,z5,tPen\WObj:=wPaper;
    MoveL Offs(pOrigin,184.07,197.80,6.00),vTravel,z5,tPen\WObj:=wPaper;
    MoveL Offs(pOrigin,184.07,197.80,0.00),v60,z0,tPen\WObj:=wPaper;
    MoveL Offs(pOrigin,186.93,200.66,0.00),v40,z0,tPen\WObj:=wPaper;
    MoveL Offs(pOrigin,186.18,201.41,0.00),v40,z0,tPen\WObj:=wPaper;
    MoveL Offs(pOrigin,192.04,207.27,0.00),v40,z0,tPen\WObj:=wPaper;
    MoveL Offs(pOrigin,191.69,207.30,0.00),v40,z0,tPen\WObj:=wPaper;
    MoveL Offs(pOrigin,196.20,202.79,0.00),v40,z0,tPen\WObj:=wPaper;
    MoveL Offs(pOrigin,195.17,202.93,0.00),v40,z0,tPen\WObj:=wPaper;
    MoveL Offs(pOrigin,197.73,205.49,0.00),v40,fine,tPen\WObj:=wPaper;
    MoveL Offs(pOrigin,197.73,205.49,6.00),v60,z5,tPen\WObj:=wPaper;
    MoveL Offs(pOrigin,198.74,206.23,6.00),vTravel,z5,tPen\WObj:=wPaper;
    MoveL Offs(pOrigin,198.74,206.23,0.00),v60,z0,tPen\WObj:=wPaper;
    MoveL Offs(pOrigin,200.84,204.12,0.00),v40,z0,tPen\WObj:=wPaper;
    MoveL Offs(pOrigin,201.62,204.90,0.00),v40,z0,tPen\WObj:=wPaper;
    MoveL Offs(pOrigin,203.57,206.85,0.00),v40,z0,tPen\WObj:=wPaper;
    MoveL Offs(pOrigin,203.68,207.26,0.00),v40,z0,tPen\WObj:=wPaper;
    MoveL Offs(pOrigin,206.23,204.71,0.00),v40,z0,tPen\WObj:=wPaper;
    MoveL Offs(pOrigin,206.56,205.36,0.00),v40,z0,tPen\WObj:=wPaper;
    MoveL Offs(pOrigin,209.12,207.92,0.00),v40,z0,tPen\WObj:=wPaper;
    MoveL Offs(pOrigin,208.77,208.14,0.00),v40,z0,tPen\WObj:=wPaper;
    MoveL Offs(pOrigin,212.07,204.84,0.00),v40,z0,tPen\WObj:=wPaper;
    MoveL Offs(pOrigin,211.11,205.08,0.00),v40,z0,tPen\WObj:=wPaper;
    MoveL Offs(pOrigin,208.99,205.08,0.00),v40,z0,tPen\WObj:=wPaper;
    MoveL Offs(pOrigin,208.35,204.32,0.00),v40,z0,tPen\WObj:=wPaper;
    MoveL Offs(pOrigin,209.20,205.18,0.00),v40,z0,tPen\WObj:=wPaper;
    MoveL Offs(pOrigin,208.35,204.32,0.00),v40,z0,tPen\WObj:=wPaper;
    MoveL Offs(pOrigin,208.35,204.02,0.00),v40,z0,tPen\WObj:=wPaper;
    MoveL Offs(pOrigin,210.05,204.02,0.00),v40,z0,tPen\WObj:=wPaper;
    MoveL Offs(pOrigin,210.48,204.32,0.00),v40,z0,tPen\WObj:=wPaper;
    MoveL Offs(pOrigin,211.32,205.18,0.00),v40,z0,tPen\WObj:=wPaper;
    MoveL Offs(pOrigin,210.48,204.32,0.00),v40,z0,tPen\WObj:=wPaper;
    MoveL Offs(pOrigin,211.32,204.09,0.00),v40,z0,tPen\WObj:=wPaper;
    MoveL Offs(pOrigin,207.57,207.85,0.00),v40,z0,tPen\WObj:=wPaper;
    MoveL Offs(pOrigin,207.02,207.31,0.00),v40,z0,tPen\WObj:=wPaper;
    MoveL Offs(pOrigin,204.92,205.21,0.00),v40,z0,tPen\WObj:=wPaper;
    MoveL Offs(pOrigin,204.73,204.71,0.00),v40,z0,tPen\WObj:=wPaper;
    MoveL Offs(pOrigin,202.48,206.97,0.00),v40,z0,tPen\WObj:=wPaper;
    MoveL Offs(pOrigin,201.62,206.40,0.00),v40,z0,tPen\WObj:=wPaper;
    MoveL Offs(pOrigin,199.67,204.44,0.00),v40,z0,tPen\WObj:=wPaper;
    MoveL Offs(pOrigin,199.79,203.68,0.00),v40,z0,tPen\WObj:=wPaper;
    MoveL Offs(pOrigin,194.68,208.79,0.00),v40,z0,tPen\WObj:=wPaper;
    MoveL Offs(pOrigin,195.19,208.92,0.00),v40,z0,tPen\WObj:=wPaper;
    MoveL Offs(pOrigin,189.18,202.91,0.00),v40,z0,tPen\WObj:=wPaper;
    MoveL Offs(pOrigin,188.38,202.97,0.00),v40,z0,tPen\WObj:=wPaper;
    MoveL Offs(pOrigin,185.40,202.97,0.00),v40,z0,tPen\WObj:=wPaper;
  ENDPROC

  PROC DrawPart115()
    MoveL Offs(pOrigin,184.55,202.84,0.00),v40,z0,tPen\WObj:=wPaper;
    MoveL Offs(pOrigin,184.98,203.05,0.00),v40,z0,tPen\WObj:=wPaper;
    MoveL Offs(pOrigin,184.55,202.84,0.00),v40,z0,tPen\WObj:=wPaper;
    MoveL Offs(pOrigin,183.91,203.13,0.00),v40,z0,tPen\WObj:=wPaper;
    MoveL Offs(pOrigin,188.12,198.92,0.00),v40,z0,tPen\WObj:=wPaper;
    MoveL Offs(pOrigin,189.02,199.52,0.00),v40,z0,tPen\WObj:=wPaper;
    MoveL Offs(pOrigin,184.81,203.72,0.00),v40,z0,tPen\WObj:=wPaper;
    MoveL Offs(pOrigin,185.86,204.17,0.00),v40,z0,tPen\WObj:=wPaper;
    MoveL Offs(pOrigin,190.07,199.96,0.00),v40,z0,tPen\WObj:=wPaper;
    MoveL Offs(pOrigin,189.77,200.52,0.00),v40,z0,tPen\WObj:=wPaper;
    MoveL Offs(pOrigin,193.08,203.82,0.00),v40,z0,tPen\WObj:=wPaper;
    MoveL Offs(pOrigin,192.33,204.57,0.00),v40,z0,tPen\WObj:=wPaper;
    MoveL Offs(pOrigin,198.04,210.28,0.00),v40,z0,tPen\WObj:=wPaper;
    MoveL Offs(pOrigin,197.67,210.28,0.00),v40,z0,tPen\WObj:=wPaper;
    MoveL Offs(pOrigin,200.08,207.87,0.00),v40,z0,tPen\WObj:=wPaper;
    MoveL Offs(pOrigin,201.13,208.32,0.00),v40,z0,tPen\WObj:=wPaper;
    MoveL Offs(pOrigin,198.72,210.72,0.00),v40,z0,tPen\WObj:=wPaper;
    MoveL Offs(pOrigin,199.77,211.17,0.00),v40,z0,tPen\WObj:=wPaper;
    MoveL Offs(pOrigin,202.17,208.76,0.00),v40,z0,tPen\WObj:=wPaper;
    MoveL Offs(pOrigin,201.33,209.09,0.00),v40,z0,tPen\WObj:=wPaper;
    MoveL Offs(pOrigin,204.79,212.55,0.00),v40,z0,tPen\WObj:=wPaper;
    MoveL Offs(pOrigin,204.26,212.65,0.00),v40,z0,tPen\WObj:=wPaper;
    MoveL Offs(pOrigin,206.66,210.25,0.00),v40,z0,tPen\WObj:=wPaper;
    MoveL Offs(pOrigin,205.83,210.60,0.00),v40,z0,tPen\WObj:=wPaper;
    MoveL Offs(pOrigin,208.69,213.46,0.00),v40,z0,tPen\WObj:=wPaper;
    MoveL Offs(pOrigin,209.20,213.69,0.00),v40,z0,tPen\WObj:=wPaper;
    MoveL Offs(pOrigin,214.91,207.98,0.00),v40,z0,tPen\WObj:=wPaper;
    MoveL Offs(pOrigin,214.09,208.36,0.00),v40,z0,tPen\WObj:=wPaper;
    MoveL Offs(pOrigin,215.79,210.06,0.00),v40,z0,tPen\WObj:=wPaper;
    MoveL Offs(pOrigin,214.09,208.36,0.00),v40,z0,tPen\WObj:=wPaper;
    MoveL Offs(pOrigin,213.88,208.25,0.00),v40,z0,tPen\WObj:=wPaper;
    MoveL Offs(pOrigin,211.32,208.25,0.00),v40,z0,tPen\WObj:=wPaper;
    MoveL Offs(pOrigin,211.21,207.94,0.00),v40,z0,tPen\WObj:=wPaper;
    MoveL Offs(pOrigin,211.21,206.02,0.00),v40,z0,tPen\WObj:=wPaper;
    MoveL Offs(pOrigin,211.75,205.81,0.00),v40,z0,tPen\WObj:=wPaper;
    MoveL Offs(pOrigin,212.60,206.66,0.00),v40,z0,tPen\WObj:=wPaper;
    MoveL Offs(pOrigin,211.75,205.81,0.00),v40,z0,tPen\WObj:=wPaper;
    MoveL Offs(pOrigin,211.96,206.14,0.00),v40,z0,tPen\WObj:=wPaper;
    MoveL Offs(pOrigin,204.74,206.14,0.00),v40,z0,tPen\WObj:=wPaper;
    MoveL Offs(pOrigin,205.07,206.86,0.00),v40,z0,tPen\WObj:=wPaper;
    MoveL Offs(pOrigin,203.12,204.90,0.00),v40,z0,tPen\WObj:=wPaper;
    MoveL Offs(pOrigin,203.53,204.42,0.00),v40,z0,tPen\WObj:=wPaper;
    MoveL Offs(pOrigin,201.28,206.67,0.00),v40,fine,tPen\WObj:=wPaper;
    MoveL Offs(pOrigin,201.28,206.67,6.00),v60,z5,tPen\WObj:=wPaper;
    MoveL Offs(pOrigin,199.93,206.52,6.00),vTravel,z5,tPen\WObj:=wPaper;
    MoveL Offs(pOrigin,199.93,206.52,0.00),v60,z0,tPen\WObj:=wPaper;
    MoveL Offs(pOrigin,202.19,204.27,0.00),v40,fine,tPen\WObj:=wPaper;
    MoveL Offs(pOrigin,202.19,204.27,6.00),v60,z5,tPen\WObj:=wPaper;
    MoveL Offs(pOrigin,199.98,206.24,6.00),vTravel,z5,tPen\WObj:=wPaper;
    MoveL Offs(pOrigin,199.98,206.24,0.00),v60,z0,tPen\WObj:=wPaper;
    MoveL Offs(pOrigin,197.57,203.84,0.00),v40,z0,tPen\WObj:=wPaper;
    MoveL Offs(pOrigin,197.55,202.94,0.00),v40,z0,tPen\WObj:=wPaper;
    MoveL Offs(pOrigin,192.74,207.74,0.00),v40,z0,tPen\WObj:=wPaper;
    MoveL Offs(pOrigin,193.48,207.51,0.00),v40,z0,tPen\WObj:=wPaper;
    MoveL Offs(pOrigin,193.90,207.73,0.00),v40,z0,tPen\WObj:=wPaper;
    MoveL Offs(pOrigin,193.48,207.51,0.00),v40,z0,tPen\WObj:=wPaper;
    MoveL Offs(pOrigin,193.48,207.19,0.00),v40,z0,tPen\WObj:=wPaper;
    MoveL Offs(pOrigin,196.45,207.19,0.00),v40,z0,tPen\WObj:=wPaper;
    MoveL Offs(pOrigin,196.88,207.51,0.00),v40,z0,tPen\WObj:=wPaper;
    MoveL Offs(pOrigin,197.30,207.73,0.00),v40,z0,tPen\WObj:=wPaper;
    MoveL Offs(pOrigin,196.88,207.51,0.00),v40,fine,tPen\WObj:=wPaper;
    MoveL Offs(pOrigin,196.88,207.51,6.00),v60,z5,tPen\WObj:=wPaper;
    MoveL Offs(pOrigin,197.98,206.98,6.00),vTravel,z5,tPen\WObj:=wPaper;
    MoveL Offs(pOrigin,197.98,206.98,0.00),v60,z0,tPen\WObj:=wPaper;
    MoveL Offs(pOrigin,195.58,209.38,0.00),v40,z0,tPen\WObj:=wPaper;
    MoveL Offs(pOrigin,195.18,208.36,0.00),v40,z0,tPen\WObj:=wPaper;
    MoveL Offs(pOrigin,195.60,208.57,0.00),v40,z0,tPen\WObj:=wPaper;
    MoveL Offs(pOrigin,195.18,208.36,0.00),v40,z0,tPen\WObj:=wPaper;
    MoveL Offs(pOrigin,195.60,208.25,0.00),v40,z0,tPen\WObj:=wPaper;
    MoveL Offs(pOrigin,198.58,208.25,0.00),v40,z0,tPen\WObj:=wPaper;
    MoveL Offs(pOrigin,198.57,208.36,0.00),v40,z0,tPen\WObj:=wPaper;
    MoveL Offs(pOrigin,199.00,208.57,0.00),v40,z0,tPen\WObj:=wPaper;
    MoveL Offs(pOrigin,198.57,208.36,0.00),v40,z0,tPen\WObj:=wPaper;
    MoveL Offs(pOrigin,198.93,208.19,0.00),v40,z0,tPen\WObj:=wPaper;
    MoveL Offs(pOrigin,202.69,211.94,0.00),v40,z0,tPen\WObj:=wPaper;
    MoveL Offs(pOrigin,203.06,212.36,0.00),v40,z0,tPen\WObj:=wPaper;
    MoveL Offs(pOrigin,205.61,209.80,0.00),v40,fine,tPen\WObj:=wPaper;
    MoveL Offs(pOrigin,205.61,209.80,6.00),v60,z5,tPen\WObj:=wPaper;
    MoveL Offs(pOrigin,204.52,210.36,6.00),vTravel,z5,tPen\WObj:=wPaper;
    MoveL Offs(pOrigin,204.52,210.36,0.00),v60,z0,tPen\WObj:=wPaper;
    MoveL Offs(pOrigin,200.49,210.36,0.00),v40,z0,tPen\WObj:=wPaper;
    MoveL Offs(pOrigin,200.59,211.34,0.00),v40,z0,tPen\WObj:=wPaper;
    MoveL Offs(pOrigin,195.78,206.53,0.00),v40,z0,tPen\WObj:=wPaper;
    MoveL Offs(pOrigin,194.75,206.45,0.00),v40,z0,tPen\WObj:=wPaper;
    MoveL Offs(pOrigin,195.18,206.66,0.00),v40,z0,tPen\WObj:=wPaper;
    MoveL Offs(pOrigin,194.75,206.45,0.00),v40,z0,tPen\WObj:=wPaper;
    MoveL Offs(pOrigin,194.32,206.14,0.00),v40,z0,tPen\WObj:=wPaper;
    MoveL Offs(pOrigin,191.56,206.14,0.00),v40,z0,tPen\WObj:=wPaper;
    MoveL Offs(pOrigin,191.56,206.45,0.00),v40,z0,tPen\WObj:=wPaper;
    MoveL Offs(pOrigin,191.99,206.66,0.00),v40,z0,tPen\WObj:=wPaper;
    MoveL Offs(pOrigin,191.56,206.45,0.00),v40,z0,tPen\WObj:=wPaper;
    MoveL Offs(pOrigin,190.71,206.02,0.00),v40,z0,tPen\WObj:=wPaper;
    MoveL Offs(pOrigin,191.14,206.24,0.00),v40,z0,tPen\WObj:=wPaper;
    MoveL Offs(pOrigin,190.71,206.02,0.00),v40,z0,tPen\WObj:=wPaper;
    MoveL Offs(pOrigin,190.64,206.85,0.00),v40,z0,tPen\WObj:=wPaper;
    MoveL Offs(pOrigin,195.15,202.34,0.00),v40,z0,tPen\WObj:=wPaper;
    MoveL Offs(pOrigin,194.25,201.75,0.00),v40,z0,tPen\WObj:=wPaper;
    MoveL Offs(pOrigin,189.75,206.26,0.00),v40,z0,tPen\WObj:=wPaper;
    MoveL Offs(pOrigin,189.86,205.60,0.00),v40,z0,tPen\WObj:=wPaper;
    MoveL Offs(pOrigin,190.29,205.81,0.00),v40,z0,tPen\WObj:=wPaper;
    MoveL Offs(pOrigin,189.86,205.60,0.00),v40,z0,tPen\WObj:=wPaper;
    MoveL Offs(pOrigin,189.44,205.08,0.00),v40,z0,tPen\WObj:=wPaper;
    MoveL Offs(pOrigin,192.41,205.08,0.00),v40,z0,tPen\WObj:=wPaper;
    MoveL Offs(pOrigin,191.99,204.96,0.00),v40,z0,tPen\WObj:=wPaper;
    MoveL Offs(pOrigin,192.41,205.18,0.00),v40,z0,tPen\WObj:=wPaper;
    MoveL Offs(pOrigin,191.99,204.96,0.00),v40,z0,tPen\WObj:=wPaper;
    MoveL Offs(pOrigin,192.84,205.39,0.00),v40,z0,tPen\WObj:=wPaper;
    MoveL Offs(pOrigin,193.48,205.81,0.00),v40,z0,tPen\WObj:=wPaper;
    MoveL Offs(pOrigin,192.84,205.39,0.00),v40,fine,tPen\WObj:=wPaper;
    MoveL Offs(pOrigin,192.84,205.39,6.00),v60,z5,tPen\WObj:=wPaper;
    MoveL Offs(pOrigin,193.90,206.02,6.00),vTravel,z5,tPen\WObj:=wPaper;
    MoveL Offs(pOrigin,193.90,206.02,0.00),v60,z0,tPen\WObj:=wPaper;
    MoveL Offs(pOrigin,194.32,206.24,0.00),v40,z0,tPen\WObj:=wPaper;
    MoveL Offs(pOrigin,193.90,206.02,0.00),v40,fine,tPen\WObj:=wPaper;
    MoveL Offs(pOrigin,193.90,206.02,6.00),v60,z5,tPen\WObj:=wPaper;
    MoveL Offs(pOrigin,195.48,204.73,6.00),vTravel,z5,tPen\WObj:=wPaper;
    MoveL Offs(pOrigin,195.48,204.73,0.00),v60,z0,tPen\WObj:=wPaper;
    MoveL Offs(pOrigin,192.77,202.03,0.00),v40,z0,tPen\WObj:=wPaper;
    MoveL Offs(pOrigin,193.06,201.45,0.00),v40,z0,tPen\WObj:=wPaper;
    MoveL Offs(pOrigin,188.85,205.66,0.00),v40,z0,tPen\WObj:=wPaper;
  ENDPROC

  PROC DrawPart116()
    MoveL Offs(pOrigin,189.04,205.76,0.00),v40,z0,tPen\WObj:=wPaper;
    MoveL Offs(pOrigin,183.48,200.20,0.00),v40,z0,tPen\WObj:=wPaper;
    MoveL Offs(pOrigin,183.06,200.50,0.00),v40,z0,tPen\WObj:=wPaper;
    MoveL Offs(pOrigin,183.49,200.71,0.00),v40,z0,tPen\WObj:=wPaper;
    MoveL Offs(pOrigin,183.06,200.50,0.00),v40,z0,tPen\WObj:=wPaper;
    MoveL Offs(pOrigin,183.91,200.86,0.00),v40,z0,tPen\WObj:=wPaper;
    MoveL Offs(pOrigin,180.94,200.86,0.00),v40,z0,tPen\WObj:=wPaper;
    MoveL Offs(pOrigin,180.77,201.79,0.00),v40,z0,tPen\WObj:=wPaper;
    MoveL Offs(pOrigin,185.13,197.43,0.00),v40,z0,tPen\WObj:=wPaper;
    MoveL Offs(pOrigin,186.03,198.03,0.00),v40,z0,tPen\WObj:=wPaper;
    MoveL Offs(pOrigin,181.67,202.39,0.00),v40,z0,tPen\WObj:=wPaper;
    MoveL Offs(pOrigin,181.79,201.56,0.00),v40,z0,tPen\WObj:=wPaper;
    MoveL Offs(pOrigin,182.21,201.77,0.00),v40,z0,tPen\WObj:=wPaper;
    MoveL Offs(pOrigin,181.79,201.56,0.00),v40,fine,tPen\WObj:=wPaper;
    MoveL Offs(pOrigin,181.79,201.56,6.00),v60,z5,tPen\WObj:=wPaper;
    MoveL Offs(pOrigin,183.06,201.91,6.00),vTravel,z5,tPen\WObj:=wPaper;
    MoveL Offs(pOrigin,183.06,201.91,0.00),v60,z0,tPen\WObj:=wPaper;
    MoveL Offs(pOrigin,186.25,201.91,0.00),v40,z0,tPen\WObj:=wPaper;
    MoveL Offs(pOrigin,185.40,201.56,0.00),v40,z0,tPen\WObj:=wPaper;
    MoveL Offs(pOrigin,185.82,201.77,0.00),v40,z0,tPen\WObj:=wPaper;
    MoveL Offs(pOrigin,185.40,201.56,0.00),v40,fine,tPen\WObj:=wPaper;
    MoveL Offs(pOrigin,185.40,201.56,6.00),v60,z5,tPen\WObj:=wPaper;
    MoveL Offs(pOrigin,187.10,202.41,6.00),vTravel,z5,tPen\WObj:=wPaper;
    MoveL Offs(pOrigin,187.10,202.41,0.00),v60,z0,tPen\WObj:=wPaper;
    MoveL Offs(pOrigin,187.52,202.62,0.00),v40,z0,tPen\WObj:=wPaper;
    MoveL Offs(pOrigin,187.10,202.41,0.00),v40,z0,tPen\WObj:=wPaper;
    MoveL Offs(pOrigin,187.95,202.84,0.00),v40,z0,tPen\WObj:=wPaper;
    MoveL Offs(pOrigin,188.38,203.05,0.00),v40,z0,tPen\WObj:=wPaper;
    MoveL Offs(pOrigin,187.95,202.84,0.00),v40,fine,tPen\WObj:=wPaper;
    MoveL Offs(pOrigin,187.95,202.84,6.00),v60,z5,tPen\WObj:=wPaper;
    MoveL Offs(pOrigin,187.52,204.02,6.00),vTravel,z5,tPen\WObj:=wPaper;
    MoveL Offs(pOrigin,187.52,204.02,0.00),v60,z0,tPen\WObj:=wPaper;
    MoveL Offs(pOrigin,190.50,204.02,0.00),v40,z0,tPen\WObj:=wPaper;
    MoveL Offs(pOrigin,190.71,204.32,0.00),v40,z0,tPen\WObj:=wPaper;
    MoveL Offs(pOrigin,191.14,204.54,0.00),v40,z0,tPen\WObj:=wPaper;
    MoveL Offs(pOrigin,190.71,204.32,0.00),v40,fine,tPen\WObj:=wPaper;
    MoveL Offs(pOrigin,190.71,204.32,6.00),v60,z5,tPen\WObj:=wPaper;
    MoveL Offs(pOrigin,190.08,202.32,6.00),vTravel,z5,tPen\WObj:=wPaper;
    MoveL Offs(pOrigin,190.08,202.32,0.00),v60,z0,tPen\WObj:=wPaper;
    MoveL Offs(pOrigin,187.07,199.31,0.00),v40,z0,tPen\WObj:=wPaper;
    MoveL Offs(pOrigin,187.07,198.47,0.00),v40,z0,tPen\WObj:=wPaper;
    MoveL Offs(pOrigin,182.87,202.68,0.00),v40,z0,tPen\WObj:=wPaper;
    MoveL Offs(pOrigin,182.89,202.59,0.00),v40,z0,tPen\WObj:=wPaper;
    MoveL Offs(pOrigin,178.38,198.09,0.00),v40,z0,tPen\WObj:=wPaper;
    MoveL Offs(pOrigin,179.02,198.74,0.00),v40,z0,tPen\WObj:=wPaper;
    MoveL Offs(pOrigin,176.05,198.74,0.00),v40,z0,tPen\WObj:=wPaper;
    MoveL Offs(pOrigin,175.54,199.56,0.00),v40,z0,tPen\WObj:=wPaper;
    MoveL Offs(pOrigin,179.74,195.35,0.00),v40,fine,tPen\WObj:=wPaper;
    MoveL Offs(pOrigin,179.74,195.35,6.00),v60,z5,tPen\WObj:=wPaper;
    MoveL Offs(pOrigin,180.94,195.65,6.00),vTravel,z5,tPen\WObj:=wPaper;
    MoveL Offs(pOrigin,180.94,195.65,0.00),v60,z0,tPen\WObj:=wPaper;
    MoveL Offs(pOrigin,176.58,200.00,0.00),v40,z0,tPen\WObj:=wPaper;
    MoveL Offs(pOrigin,177.34,200.03,0.00),v40,z0,tPen\WObj:=wPaper;
    MoveL Offs(pOrigin,173.43,196.12,0.00),v40,z0,tPen\WObj:=wPaper;
    MoveL Offs(pOrigin,173.92,196.63,0.00),v40,z0,tPen\WObj:=wPaper;
    MoveL Offs(pOrigin,170.31,196.63,0.00),v40,fine,tPen\WObj:=wPaper;
    MoveL Offs(pOrigin,170.31,196.63,6.00),v60,z5,tPen\WObj:=wPaper;
    MoveL Offs(pOrigin,169.85,197.78,6.00),vTravel,z5,tPen\WObj:=wPaper;
    MoveL Offs(pOrigin,169.85,197.78,0.00),v60,z0,tPen\WObj:=wPaper;
    MoveL Offs(pOrigin,174.36,193.27,0.00),v40,fine,tPen\WObj:=wPaper;
    MoveL Offs(pOrigin,174.36,193.27,6.00),v60,z5,tPen\WObj:=wPaper;
    MoveL Offs(pOrigin,175.56,193.57,6.00),vTravel,z5,tPen\WObj:=wPaper;
    MoveL Offs(pOrigin,175.56,193.57,0.00),v60,z0,tPen\WObj:=wPaper;
    MoveL Offs(pOrigin,169.54,199.58,0.00),v40,z0,tPen\WObj:=wPaper;
    MoveL Offs(pOrigin,170.00,200.16,0.00),v40,z0,tPen\WObj:=wPaper;
    MoveL Offs(pOrigin,171.65,201.81,0.00),v40,z0,tPen\WObj:=wPaper;
    MoveL Offs(pOrigin,171.16,201.91,0.00),v40,z0,tPen\WObj:=wPaper;
    MoveL Offs(pOrigin,170.10,201.91,0.00),v40,z0,tPen\WObj:=wPaper;
    MoveL Offs(pOrigin,169.70,201.36,0.00),v40,z0,tPen\WObj:=wPaper;
    MoveL Offs(pOrigin,171.35,203.01,0.00),v40,z0,tPen\WObj:=wPaper;
    MoveL Offs(pOrigin,171.78,203.31,0.00),v40,z0,tPen\WObj:=wPaper;
    MoveL Offs(pOrigin,167.57,207.52,0.00),v40,z0,tPen\WObj:=wPaper;
    MoveL Offs(pOrigin,168.37,207.49,0.00),v40,z0,tPen\WObj:=wPaper;
    MoveL Offs(pOrigin,170.02,209.15,0.00),v40,z0,tPen\WObj:=wPaper;
    MoveL Offs(pOrigin,170.71,208.86,0.00),v40,z0,tPen\WObj:=wPaper;
    MoveL Offs(pOrigin,163.80,215.77,0.00),v40,z0,tPen\WObj:=wPaper;
    MoveL Offs(pOrigin,164.35,215.42,0.00),v40,z0,tPen\WObj:=wPaper;
    MoveL Offs(pOrigin,166.45,217.52,0.00),v40,fine,tPen\WObj:=wPaper;
    MoveL Offs(pOrigin,166.45,217.52,6.00),v60,z5,tPen\WObj:=wPaper;
    MoveL Offs(pOrigin,166.61,219.17,6.00),vTravel,z5,tPen\WObj:=wPaper;
    MoveL Offs(pOrigin,166.61,219.17,0.00),v60,z0,tPen\WObj:=wPaper;
    MoveL Offs(pOrigin,164.36,216.92,0.00),v40,z0,tPen\WObj:=wPaper;
    MoveL Offs(pOrigin,163.80,217.27,0.00),v40,z0,tPen\WObj:=wPaper;
    MoveL Offs(pOrigin,170.41,210.66,0.00),v40,z0,tPen\WObj:=wPaper;
    MoveL Offs(pOrigin,169.88,210.49,0.00),v40,z0,tPen\WObj:=wPaper;
    MoveL Offs(pOrigin,168.08,208.69,0.00),v40,z0,tPen\WObj:=wPaper;
    MoveL Offs(pOrigin,167.42,209.17,0.00),v40,z0,tPen\WObj:=wPaper;
    MoveL Offs(pOrigin,171.32,205.26,0.00),v40,z0,tPen\WObj:=wPaper;
    MoveL Offs(pOrigin,170.76,205.40,0.00),v40,z0,tPen\WObj:=wPaper;
    MoveL Offs(pOrigin,169.11,203.75,0.00),v40,z0,tPen\WObj:=wPaper;
    MoveL Offs(pOrigin,168.48,203.62,0.00),v40,z0,tPen\WObj:=wPaper;
    MoveL Offs(pOrigin,177.65,194.46,0.00),v40,z0,tPen\WObj:=wPaper;
    MoveL Offs(pOrigin,176.87,195.09,0.00),v40,z0,tPen\WObj:=wPaper;
    MoveL Offs(pOrigin,177.77,195.99,0.00),v40,fine,tPen\WObj:=wPaper;
    MoveL Offs(pOrigin,177.77,195.99,6.00),v60,z5,tPen\WObj:=wPaper;
    MoveL Offs(pOrigin,176.48,197.69,6.00),vTravel,z5,tPen\WObj:=wPaper;
    MoveL Offs(pOrigin,176.48,197.69,0.00),v60,z0,tPen\WObj:=wPaper;
    MoveL Offs(pOrigin,171.16,197.69,0.00),v40,z0,tPen\WObj:=wPaper;
    MoveL Offs(pOrigin,170.95,198.74,0.00),v40,z0,tPen\WObj:=wPaper;
    MoveL Offs(pOrigin,172.23,198.74,0.00),v40,z0,tPen\WObj:=wPaper;
    MoveL Offs(pOrigin,172.14,198.16,0.00),v40,z0,tPen\WObj:=wPaper;
    MoveL Offs(pOrigin,172.14,196.46,0.00),v40,fine,tPen\WObj:=wPaper;
    MoveL Offs(pOrigin,172.14,196.46,6.00),v60,z5,tPen\WObj:=wPaper;
    MoveL Offs(pOrigin,172.99,198.67,6.00),vTravel,z5,tPen\WObj:=wPaper;
    MoveL Offs(pOrigin,172.99,198.67,0.00),v60,z0,tPen\WObj:=wPaper;
    MoveL Offs(pOrigin,168.48,194.16,0.00),v40,z0,tPen\WObj:=wPaper;
    MoveL Offs(pOrigin,168.19,194.52,0.00),v40,z0,tPen\WObj:=wPaper;
    MoveL Offs(pOrigin,164.15,194.52,0.00),v40,z0,tPen\WObj:=wPaper;
    MoveL Offs(pOrigin,163.24,194.89,0.00),v40,z0,tPen\WObj:=wPaper;
    MoveL Offs(pOrigin,159.93,191.59,0.00),v40,fine,tPen\WObj:=wPaper;
    MoveL Offs(pOrigin,159.93,191.59,6.00),v60,z5,tPen\WObj:=wPaper;
    MoveL Offs(pOrigin,160.53,192.85,6.00),vTravel,z5,tPen\WObj:=wPaper;
    MoveL Offs(pOrigin,160.53,192.85,0.00),v60,z0,tPen\WObj:=wPaper;
    MoveL Offs(pOrigin,160.53,194.55,0.00),v40,z0,tPen\WObj:=wPaper;
    MoveL Offs(pOrigin,161.18,194.52,0.00),v40,z0,tPen\WObj:=wPaper;
    MoveL Offs(pOrigin,159.69,194.52,0.00),v40,z0,tPen\WObj:=wPaper;
    MoveL Offs(pOrigin,159.69,195.58,0.00),v40,z0,tPen\WObj:=wPaper;
    MoveL Offs(pOrigin,160.96,195.58,0.00),v40,z0,tPen\WObj:=wPaper;
    MoveL Offs(pOrigin,161.30,195.94,0.00),v40,z0,tPen\WObj:=wPaper;
    MoveL Offs(pOrigin,155.89,190.53,0.00),v40,z0,tPen\WObj:=wPaper;
  ENDPROC

  PROC DrawPart117()
    MoveL Offs(pOrigin,156.54,190.18,0.00),v40,z0,tPen\WObj:=wPaper;
    MoveL Offs(pOrigin,154.44,192.28,0.00),v40,z0,tPen\WObj:=wPaper;
    MoveL Offs(pOrigin,154.39,192.02,0.00),v40,z0,tPen\WObj:=wPaper;
    MoveL Offs(pOrigin,151.69,189.32,0.00),v40,z0,tPen\WObj:=wPaper;
    MoveL Offs(pOrigin,152.05,188.69,0.00),v40,z0,tPen\WObj:=wPaper;
    MoveL Offs(pOrigin,149.65,191.10,0.00),v40,z0,tPen\WObj:=wPaper;
    MoveL Offs(pOrigin,150.19,190.81,0.00),v40,z0,tPen\WObj:=wPaper;
    MoveL Offs(pOrigin,147.19,187.80,0.00),v40,z0,tPen\WObj:=wPaper;
    MoveL Offs(pOrigin,147.15,188.18,0.00),v40,z0,tPen\WObj:=wPaper;
    MoveL Offs(pOrigin,144.39,188.18,0.00),v40,z0,tPen\WObj:=wPaper;
    MoveL Offs(pOrigin,143.60,188.69,0.00),v40,z0,tPen\WObj:=wPaper;
    MoveL Offs(pOrigin,138.64,183.73,0.00),v40,z0,tPen\WObj:=wPaper;
    MoveL Offs(pOrigin,137.99,183.35,0.00),v40,z0,tPen\WObj:=wPaper;
    MoveL Offs(pOrigin,140.24,181.09,0.00),v40,z0,tPen\WObj:=wPaper;
    MoveL Offs(pOrigin,139.50,181.85,0.00),v40,z0,tPen\WObj:=wPaper;
    MoveL Offs(pOrigin,138.44,181.85,0.00),v40,z0,tPen\WObj:=wPaper;
    MoveL Offs(pOrigin,137.54,182.30,0.00),v40,z0,tPen\WObj:=wPaper;
    MoveL Offs(pOrigin,139.94,179.89,0.00),v40,z0,tPen\WObj:=wPaper;
    MoveL Offs(pOrigin,139.23,179.84,0.00),v40,z0,tPen\WObj:=wPaper;
    MoveL Offs(pOrigin,136.67,177.29,0.00),v40,z0,tPen\WObj:=wPaper;
    MoveL Offs(pOrigin,136.21,177.66,0.00),v40,z0,tPen\WObj:=wPaper;
    MoveL Offs(pOrigin,138.91,174.95,0.00),v40,z0,tPen\WObj:=wPaper;
    MoveL Offs(pOrigin,138.16,174.30,0.00),v40,z0,tPen\WObj:=wPaper;
    MoveL Offs(pOrigin,135.15,171.29,0.00),v40,z0,tPen\WObj:=wPaper;
    MoveL Offs(pOrigin,135.68,171.29,0.00),v40,z0,tPen\WObj:=wPaper;
    MoveL Offs(pOrigin,136.95,171.29,0.00),v40,z0,tPen\WObj:=wPaper;
    MoveL Offs(pOrigin,138.02,171.36,0.00),v40,z0,tPen\WObj:=wPaper;
    MoveL Offs(pOrigin,135.62,173.77,0.00),v40,z0,tPen\WObj:=wPaper;
    MoveL Offs(pOrigin,135.76,173.39,0.00),v40,z0,tPen\WObj:=wPaper;
    MoveL Offs(pOrigin,138.62,176.24,0.00),v40,z0,tPen\WObj:=wPaper;
    MoveL Offs(pOrigin,139.06,176.30,0.00),v40,z0,tPen\WObj:=wPaper;
    MoveL Offs(pOrigin,136.50,178.86,0.00),v40,z0,tPen\WObj:=wPaper;
    MoveL Offs(pOrigin,137.13,179.24,0.00),v40,z0,tPen\WObj:=wPaper;
    MoveL Offs(pOrigin,140.13,182.24,0.00),v40,z0,tPen\WObj:=wPaper;
    MoveL Offs(pOrigin,140.14,182.65,0.00),v40,z0,tPen\WObj:=wPaper;
    MoveL Offs(pOrigin,140.35,183.07,0.00),v40,z0,tPen\WObj:=wPaper;
    MoveL Offs(pOrigin,140.14,182.65,0.00),v40,z0,tPen\WObj:=wPaper;
    MoveL Offs(pOrigin,139.93,182.90,0.00),v40,z0,tPen\WObj:=wPaper;
    MoveL Offs(pOrigin,138.86,182.90,0.00),v40,fine,tPen\WObj:=wPaper;
    MoveL Offs(pOrigin,138.86,182.90,6.00),v60,z5,tPen\WObj:=wPaper;
    MoveL Offs(pOrigin,139.50,183.96,6.00),vTravel,z5,tPen\WObj:=wPaper;
    MoveL Offs(pOrigin,139.50,183.96,0.00),v60,z0,tPen\WObj:=wPaper;
    MoveL Offs(pOrigin,140.56,183.96,0.00),v40,z0,tPen\WObj:=wPaper;
    MoveL Offs(pOrigin,141.13,183.19,0.00),v40,z0,tPen\WObj:=wPaper;
    MoveL Offs(pOrigin,139.03,185.29,0.00),v40,z0,tPen\WObj:=wPaper;
    MoveL Offs(pOrigin,139.29,184.77,0.00),v40,z0,tPen\WObj:=wPaper;
    MoveL Offs(pOrigin,139.93,185.62,0.00),v40,z0,tPen\WObj:=wPaper;
    MoveL Offs(pOrigin,139.29,184.77,0.00),v40,z0,tPen\WObj:=wPaper;
    MoveL Offs(pOrigin,140.14,185.02,0.00),v40,z0,tPen\WObj:=wPaper;
    MoveL Offs(pOrigin,141.20,185.02,0.00),v40,z0,tPen\WObj:=wPaper;
    MoveL Offs(pOrigin,141.84,185.20,0.00),v40,z0,tPen\WObj:=wPaper;
    MoveL Offs(pOrigin,142.26,185.62,0.00),v40,z0,tPen\WObj:=wPaper;
    MoveL Offs(pOrigin,141.84,185.20,0.00),v40,z0,tPen\WObj:=wPaper;
    MoveL Offs(pOrigin,142.48,184.83,0.00),v40,z0,tPen\WObj:=wPaper;
    MoveL Offs(pOrigin,140.22,187.08,0.00),v40,z0,tPen\WObj:=wPaper;
    MoveL Offs(pOrigin,140.77,186.69,0.00),v40,z0,tPen\WObj:=wPaper;
    MoveL Offs(pOrigin,141.41,187.32,0.00),v40,z0,tPen\WObj:=wPaper;
    MoveL Offs(pOrigin,140.77,186.69,0.00),v40,z0,tPen\WObj:=wPaper;
    MoveL Offs(pOrigin,140.99,186.07,0.00),v40,z0,tPen\WObj:=wPaper;
    MoveL Offs(pOrigin,142.48,186.07,0.00),v40,z0,tPen\WObj:=wPaper;
    MoveL Offs(pOrigin,142.26,187.13,0.00),v40,z0,tPen\WObj:=wPaper;
    MoveL Offs(pOrigin,145.66,187.13,0.00),v40,z0,tPen\WObj:=wPaper;
    MoveL Offs(pOrigin,145.69,186.30,0.00),v40,z0,tPen\WObj:=wPaper;
    MoveL Offs(pOrigin,144.18,184.80,0.00),v40,z0,tPen\WObj:=wPaper;
    MoveL Offs(pOrigin,143.74,185.85,0.00),v40,z0,tPen\WObj:=wPaper;
    MoveL Offs(pOrigin,148.10,190.20,0.00),v40,z0,tPen\WObj:=wPaper;
    MoveL Offs(pOrigin,148.60,190.65,0.00),v40,z0,tPen\WObj:=wPaper;
    MoveL Offs(pOrigin,150.85,188.40,0.00),v40,z0,tPen\WObj:=wPaper;
    MoveL Offs(pOrigin,150.34,189.24,0.00),v40,z0,tPen\WObj:=wPaper;
    MoveL Offs(pOrigin,147.79,189.24,0.00),v40,z0,tPen\WObj:=wPaper;
    MoveL Offs(pOrigin,147.40,190.36,0.00),v40,z0,tPen\WObj:=wPaper;
    MoveL Offs(pOrigin,149.81,187.95,0.00),v40,z0,tPen\WObj:=wPaper;
    MoveL Offs(pOrigin,149.44,188.56,0.00),v40,z0,tPen\WObj:=wPaper;
    MoveL Offs(pOrigin,152.59,191.72,0.00),v40,z0,tPen\WObj:=wPaper;
    MoveL Offs(pOrigin,152.04,191.69,0.00),v40,z0,tPen\WObj:=wPaper;
    MoveL Offs(pOrigin,154.30,189.44,0.00),v40,z0,tPen\WObj:=wPaper;
    MoveL Offs(pOrigin,153.79,189.92,0.00),v40,z0,tPen\WObj:=wPaper;
    MoveL Offs(pOrigin,156.64,192.78,0.00),v40,z0,tPen\WObj:=wPaper;
    MoveL Offs(pOrigin,156.68,193.02,0.00),v40,z0,tPen\WObj:=wPaper;
    MoveL Offs(pOrigin,159.69,190.02,0.00),v40,fine,tPen\WObj:=wPaper;
    MoveL Offs(pOrigin,159.69,190.02,6.00),v60,z5,tPen\WObj:=wPaper;
    MoveL Offs(pOrigin,158.41,189.66,6.00),vTravel,z5,tPen\WObj:=wPaper;
    MoveL Offs(pOrigin,158.41,189.66,0.00),v60,z0,tPen\WObj:=wPaper;
    MoveL Offs(pOrigin,177.32,195.33,0.00),v40,z0,tPen\WObj:=wPaper;
    MoveL Offs(pOrigin,181.57,197.03,0.00),v40,z0,tPen\WObj:=wPaper;
    MoveL Offs(pOrigin,190.50,201.35,0.00),v40,z0,tPen\WObj:=wPaper;
    MoveL Offs(pOrigin,190.96,200.56,0.00),v40,z0,tPen\WObj:=wPaper;
    MoveL Offs(pOrigin,186.91,204.62,0.00),v40,z0,tPen\WObj:=wPaper;
    MoveL Offs(pOrigin,187.52,204.32,0.00),v40,z0,tPen\WObj:=wPaper;
    MoveL Offs(pOrigin,187.95,204.54,0.00),v40,z0,tPen\WObj:=wPaper;
    MoveL Offs(pOrigin,187.52,204.32,0.00),v40,z0,tPen\WObj:=wPaper;
    MoveL Offs(pOrigin,187.80,205.21,0.00),v40,z0,tPen\WObj:=wPaper;
    MoveL Offs(pOrigin,192.16,200.86,0.00),v40,fine,tPen\WObj:=wPaper;
    MoveL Offs(pOrigin,192.16,200.86,6.00),v60,z5,tPen\WObj:=wPaper;
    MoveL Offs(pOrigin,189.01,200.93,6.00),vTravel,z5,tPen\WObj:=wPaper;
    MoveL Offs(pOrigin,189.01,200.93,0.00),v60,z0,tPen\WObj:=wPaper;
    MoveL Offs(pOrigin,189.44,201.14,0.00),v40,z0,tPen\WObj:=wPaper;
    MoveL Offs(pOrigin,189.01,200.93,0.00),v40,fine,tPen\WObj:=wPaper;
    MoveL Offs(pOrigin,189.01,200.93,6.00),v60,z5,tPen\WObj:=wPaper;
    MoveL Offs(pOrigin,185.89,204.10,6.00),vTravel,z5,tPen\WObj:=wPaper;
    MoveL Offs(pOrigin,185.89,204.10,0.00),v60,z0,tPen\WObj:=wPaper;
    MoveL Offs(pOrigin,180.93,199.14,0.00),v40,z0,tPen\WObj:=wPaper;
    MoveL Offs(pOrigin,181.58,199.80,0.00),v40,z0,tPen\WObj:=wPaper;
    MoveL Offs(pOrigin,178.60,199.80,0.00),v40,z0,tPen\WObj:=wPaper;
    MoveL Offs(pOrigin,178.68,200.90,0.00),v40,z0,tPen\WObj:=wPaper;
    MoveL Offs(pOrigin,183.04,196.54,0.00),v40,z0,tPen\WObj:=wPaper;
    MoveL Offs(pOrigin,181.99,196.09,0.00),v40,z0,tPen\WObj:=wPaper;
    MoveL Offs(pOrigin,177.63,200.45,0.00),v40,fine,tPen\WObj:=wPaper;
    MoveL Offs(pOrigin,177.63,200.45,6.00),v60,z5,tPen\WObj:=wPaper;
    MoveL Offs(pOrigin,179.73,201.34,6.00),vTravel,z5,tPen\WObj:=wPaper;
    MoveL Offs(pOrigin,179.73,201.34,0.00),v60,z0,tPen\WObj:=wPaper;
    MoveL Offs(pOrigin,184.08,196.99,0.00),v40,fine,tPen\WObj:=wPaper;
    MoveL Offs(pOrigin,184.08,196.99,6.00),v60,z5,tPen\WObj:=wPaper;
    MoveL Offs(pOrigin,183.49,202.41,6.00),vTravel,z5,tPen\WObj:=wPaper;
    MoveL Offs(pOrigin,183.49,202.41,0.00),v60,z0,tPen\WObj:=wPaper;
    MoveL Offs(pOrigin,183.91,202.62,0.00),v40,z0,tPen\WObj:=wPaper;
    MoveL Offs(pOrigin,183.49,202.41,0.00),v40,fine,tPen\WObj:=wPaper;
    MoveL Offs(pOrigin,183.49,202.41,6.00),v60,z5,tPen\WObj:=wPaper;
    MoveL Offs(pOrigin,179.89,201.09,6.00),vTravel,z5,tPen\WObj:=wPaper;
    MoveL Offs(pOrigin,179.89,201.09,0.00),v60,z0,tPen\WObj:=wPaper;
  ENDPROC

